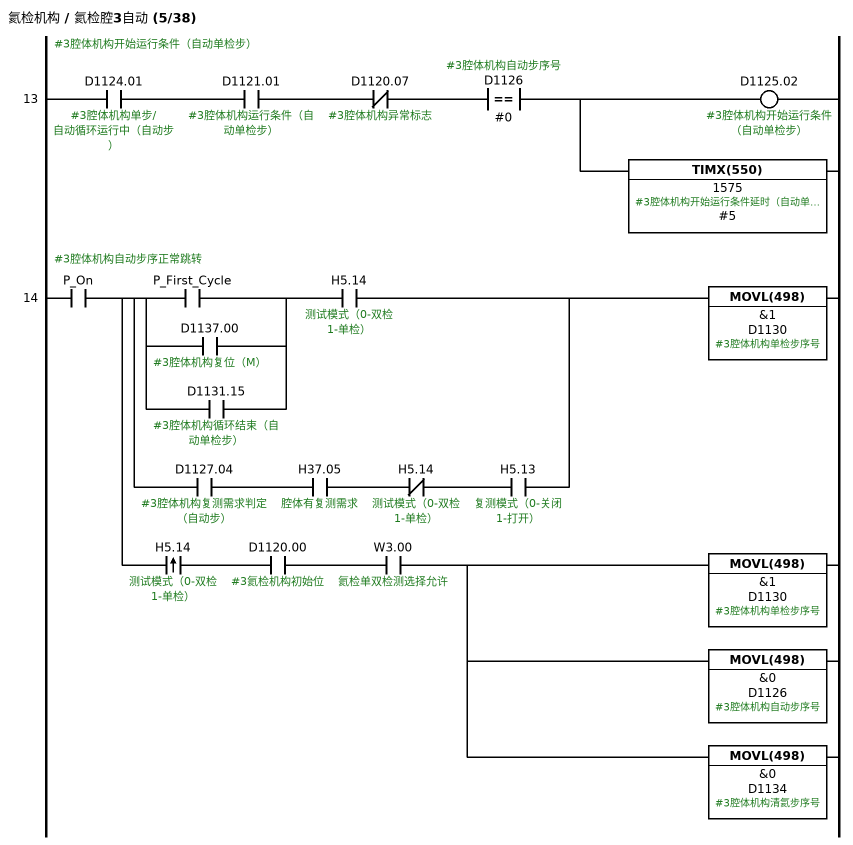
; [picture p288: 氦检机构 / 氦检腔3自动, rungs 13-14]
; rung 13: #3腔体机构开始运行条件（自动单检步）
LD D1124.01  ; #3腔体机构单步/自动循环运行中（自动步）
AND D1121.01  ; #3腔体机构运行条件（自动单检步）
ANDNOT D1120.07  ; #3腔体机构异常标志
AND=L(301) D1126 #0  ; #3腔体机构自动步序号
OUT D1125.02  ; #3腔体机构开始运行条件（自动单检步）
TIMX(550) 1575 #5  ; #3腔体机构开始运行条件延时（自动单检步）
; rung 14: #3腔体机构自动步序正常跳转
LD P_On
OUT TR0
LD P_First_Cycle
OR D1137.00  ; #3腔体机构复位（M）
OR D1131.15  ; #3腔体机构循环结束（自动单检步）
AND H5.14  ; 测试模式（0-双检 1-单检）
LD D1127.04  ; #3腔体机构复测需求判定（自动步）
AND H37.05  ; 腔体有复测需求
ANDNOT H5.14  ; 测试模式（0-双检 1-单检）
AND H5.13  ; 复测模式（0-关闭 1-打开）
ORLD
ANDLD
MOVL(498) &1 D1130  ; #3腔体机构单检步序号
LD TR0
@AND H5.14  ; 测试模式（0-双检 1-单检）
AND D1120.00  ; #3氦检机构初始位
AND W3.00  ; 氦检单双检测选择允许
MOVL(498) &1 D1130  ; #3腔体机构单检步序号
MOVL(498) &0 D1126  ; #3腔体机构自动步序号
MOVL(498) &0 D1134  ; #3腔体机构清氦步序号

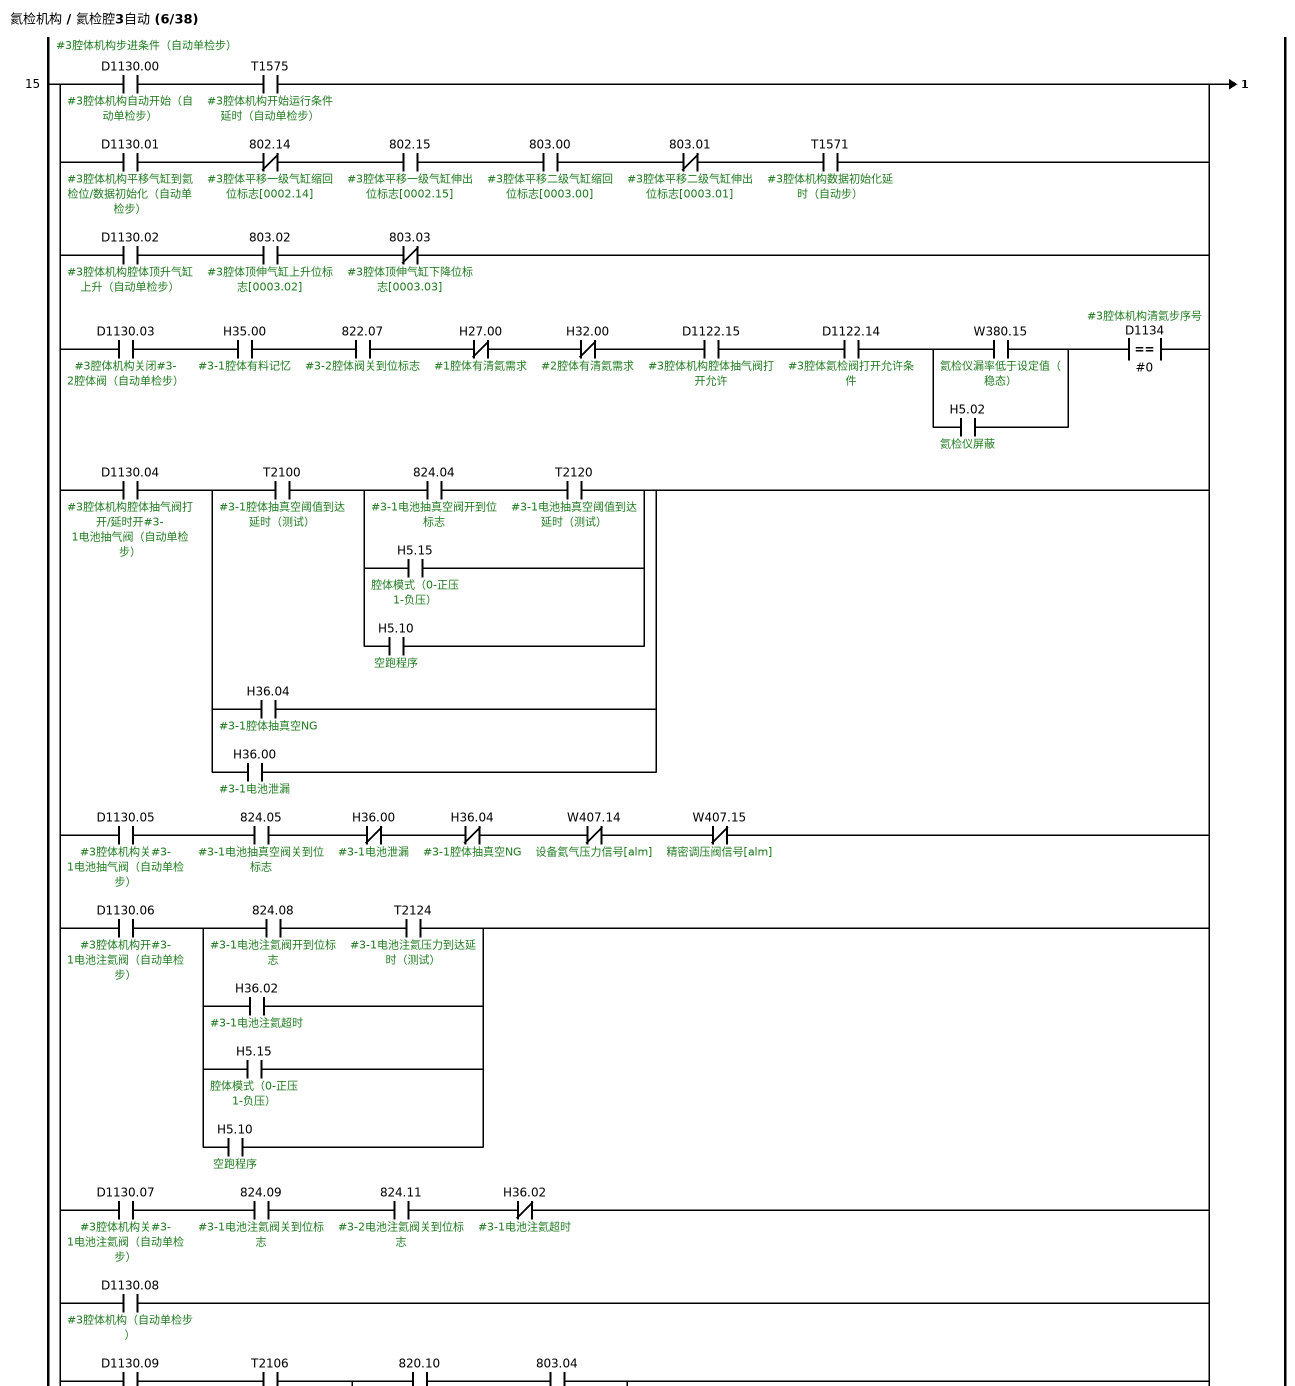

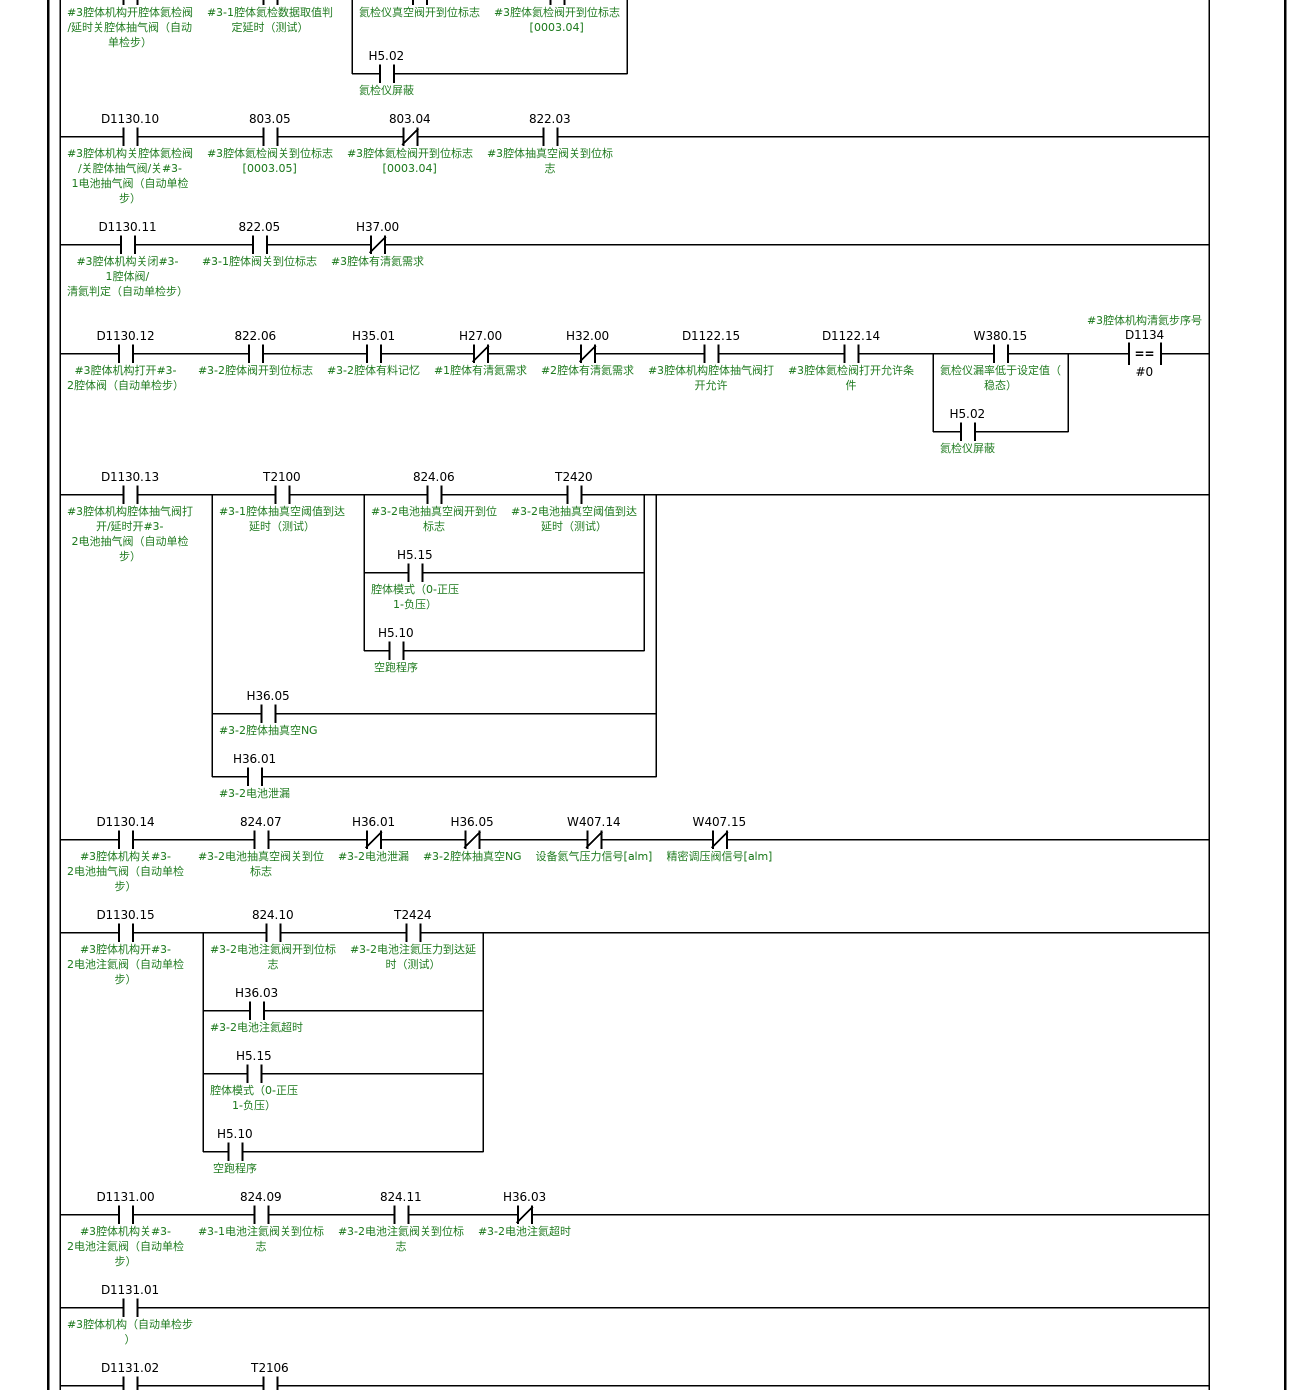

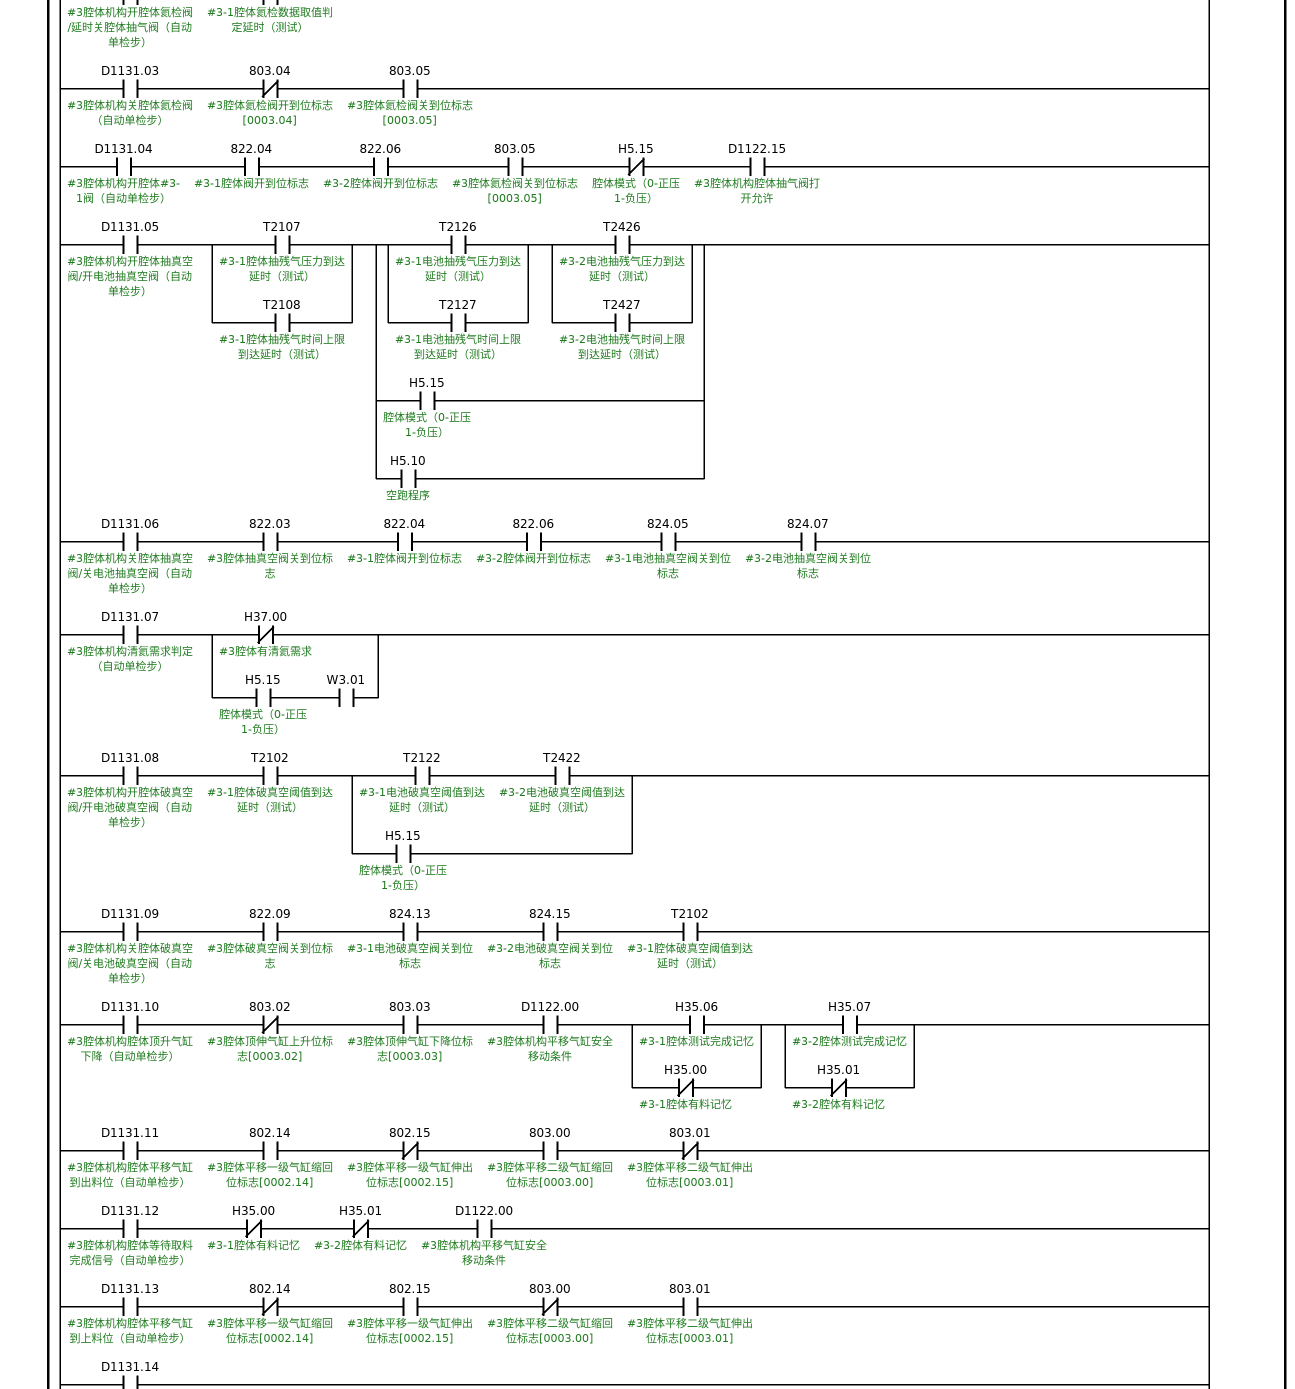

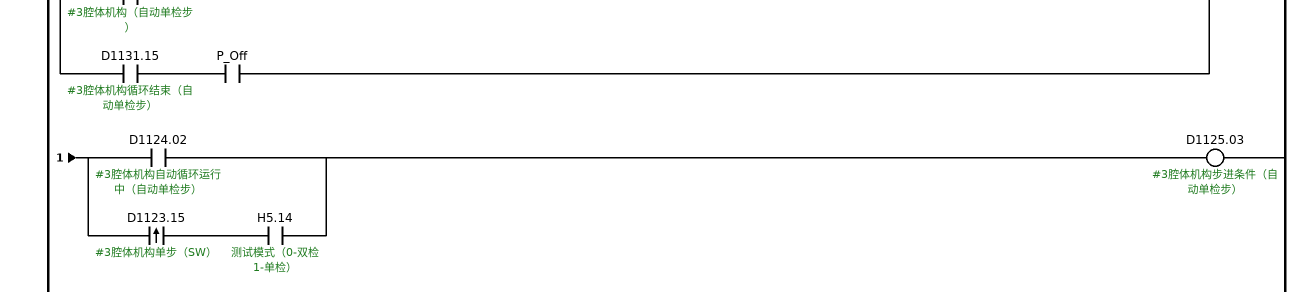
; rung 15: #3腔体机构步进条件（自动单检步）
LD D1130.00  ; #3腔体机构自动开始（自动单检步）
AND T1575  ; #3腔体机构开始运行条件延时（自动单检步）
LD D1130.01  ; #3腔体机构平移气缸到氦检位/数据初始化（自动单检步）
ANDNOT 802.14  ; #3腔体平移一级气缸缩回位标志[0002.14]
AND 802.15  ; #3腔体平移一级气缸伸出位标志[0002.15]
AND 803.00  ; #3腔体平移二级气缸缩回位标志[0003.00]
ANDNOT 803.01  ; #3腔体平移二级气缸伸出位标志[0003.01]
AND T1571  ; #3腔体机构数据初始化延时（自动步）
ORLD
LD D1130.02  ; #3腔体机构腔体顶升气缸上升（自动单检步）
AND 803.02  ; #3腔体顶伸气缸上升位标志[0003.02]
ANDNOT 803.03  ; #3腔体顶伸气缸下降位标志[0003.03]
ORLD
LD D1130.03  ; #3腔体机构关闭#3-2腔体阀（自动单检步）
AND H35.00  ; #3-1腔体有料记忆
AND 822.07  ; #3-2腔体阀关到位标志
ANDNOT H27.00  ; #1腔体有清氦需求
ANDNOT H32.00  ; #2腔体有清氦需求
AND D1122.15  ; #3腔体机构腔体抽气阀打开允许
AND D1122.14  ; #3腔体氦检阀打开允许条件
LD W380.15  ; 氦检仪漏率低于设定值（稳态）
OR H5.02  ; 氦检仪屏蔽
ANDLD
AND=L(301) D1134 #0  ; #3腔体机构清氦步序号
ORLD
LD D1130.04  ; #3腔体机构腔体抽气阀打开/延时开#3-1电池抽气阀（自动单检步）
LD T2100  ; #3-1腔体抽真空阈值到达延时（测试）
LD 824.04  ; #3-1电池抽真空阀开到位标志
AND T2120  ; #3-1电池抽真空阈值到达延时（测试）
OR H5.15  ; 腔体模式（0-正压 1-负压）
OR H5.10  ; 空跑程序
ANDLD
OR H36.04  ; #3-1腔体抽真空NG
OR H36.00  ; #3-1电池泄漏
ANDLD
ORLD
LD D1130.05  ; #3腔体机构关#3-1电池抽气阀（自动单检步）
AND 824.05  ; #3-1电池抽真空阀关到位标志
ANDNOT H36.00  ; #3-1电池泄漏
ANDNOT H36.04  ; #3-1腔体抽真空NG
ANDNOT W407.14  ; 设备氦气压力信号[alm]
ANDNOT W407.15  ; 精密调压阀信号[alm]
ORLD
LD D1130.06  ; #3腔体机构开#3-1电池注氦阀（自动单检步）
LD 824.08  ; #3-1电池注氦阀开到位标志
AND T2124  ; #3-1电池注氦压力到达延时（测试）
OR H36.02  ; #3-1电池注氦超时
OR H5.15  ; 腔体模式（0-正压 1-负压）
OR H5.10  ; 空跑程序
ANDLD
ORLD
LD D1130.07  ; #3腔体机构关#3-1电池注氦阀（自动单检步）
AND 824.09  ; #3-1电池注氦阀关到位标志
AND 824.11  ; #3-2电池注氦阀关到位标志
ANDNOT H36.02  ; #3-1电池注氦超时
ORLD
OR D1130.08  ; #3腔体机构（自动单检步）
LD D1130.09  ; #3腔体机构开腔体氦检阀/延时关腔体抽气阀（自动单检步）
AND T2106  ; #3-1腔体氦检数据取值判定延时（测试）
LD 820.10  ; 氦检仪真空阀开到位标志
AND 803.04  ; #3腔体氦检阀开到位标志[0003.04]
OR H5.02  ; 氦检仪屏蔽
ANDLD
ORLD
LD D1130.10  ; #3腔体机构关腔体氦检阀/关腔体抽气阀/关#3-1电池抽气阀（自动单检步）
AND 803.05  ; #3腔体氦检阀关到位标志[0003.05]
ANDNOT 803.04  ; #3腔体氦检阀开到位标志[0003.04]
AND 822.03  ; #3腔体抽真空阀关到位标志
ORLD
LD D1130.11  ; #3腔体机构关闭#3-1腔体阀/清氦判定（自动单检步）
AND 822.05  ; #3-1腔体阀关到位标志
ANDNOT H37.00  ; #3腔体有清氦需求
ORLD
LD D1130.12  ; #3腔体机构打开#3-2腔体阀（自动单检步）
AND 822.06  ; #3-2腔体阀开到位标志
AND H35.01  ; #3-2腔体有料记忆
ANDNOT H27.00  ; #1腔体有清氦需求
ANDNOT H32.00  ; #2腔体有清氦需求
AND D1122.15  ; #3腔体机构腔体抽气阀打开允许
AND D1122.14  ; #3腔体氦检阀打开允许条件
LD W380.15  ; 氦检仪漏率低于设定值（稳态）
OR H5.02  ; 氦检仪屏蔽
ANDLD
AND=L(301) D1134 #0  ; #3腔体机构清氦步序号
ORLD
LD D1130.13  ; #3腔体机构腔体抽气阀打开/延时开#3-2电池抽气阀（自动单检步）
LD T2100  ; #3-1腔体抽真空阈值到达延时（测试）
LD 824.06  ; #3-2电池抽真空阀开到位标志
AND T2420  ; #3-2电池抽真空阈值到达延时（测试）
OR H5.15  ; 腔体模式（0-正压 1-负压）
OR H5.10  ; 空跑程序
ANDLD
OR H36.05  ; #3-2腔体抽真空NG
OR H36.01  ; #3-2电池泄漏
ANDLD
ORLD
LD D1130.14  ; #3腔体机构关#3-2电池抽气阀（自动单检步）
AND 824.07  ; #3-2电池抽真空阀关到位标志
ANDNOT H36.01  ; #3-2电池泄漏
ANDNOT H36.05  ; #3-2腔体抽真空NG
ANDNOT W407.14  ; 设备氦气压力信号[alm]
ANDNOT W407.15  ; 精密调压阀信号[alm]
ORLD
LD D1130.15  ; #3腔体机构开#3-2电池注氦阀（自动单检步）
LD 824.10  ; #3-2电池注氦阀开到位标志
AND T2424  ; #3-2电池注氦压力到达延时（测试）
OR H36.03  ; #3-2电池注氦超时
OR H5.15  ; 腔体模式（0-正压 1-负压）
OR H5.10  ; 空跑程序
ANDLD
ORLD
LD D1131.00  ; #3腔体机构关#3-2电池注氦阀（自动单检步）
AND 824.09  ; #3-1电池注氦阀关到位标志
AND 824.11  ; #3-2电池注氦阀关到位标志
ANDNOT H36.03  ; #3-2电池注氦超时
ORLD
OR D1131.01  ; #3腔体机构（自动单检步）
LD D1131.02  ; #3腔体机构开腔体氦检阀/延时关腔体抽气阀（自动单检步）
AND T2106  ; #3-1腔体氦检数据取值判定延时（测试）
ORLD
LD D1131.03  ; #3腔体机构关腔体氦检阀（自动单检步）
ANDNOT 803.04  ; #3腔体氦检阀开到位标志[0003.04]
AND 803.05  ; #3腔体氦检阀关到位标志[0003.05]
ORLD
LD D1131.04  ; #3腔体机构开腔体#3-1阀（自动单检步）
AND 822.04  ; #3-1腔体阀开到位标志
AND 822.06  ; #3-2腔体阀开到位标志
AND 803.05  ; #3腔体氦检阀关到位标志[0003.05]
ANDNOT H5.15  ; 腔体模式（0-正压 1-负压）
AND D1122.15  ; #3腔体机构腔体抽气阀打开允许
ORLD
LD D1131.05  ; #3腔体机构开腔体抽真空阀/开电池抽真空阀（自动单检步）
LD T2107  ; #3-1腔体抽残气压力到达延时（测试）
OR T2108  ; #3-1腔体抽残气时间上限到达延时（测试）
ANDLD
LD T2126  ; #3-1电池抽残气压力到达延时（测试）
OR T2127  ; #3-1电池抽残气时间上限到达延时（测试）
LD T2426  ; #3-2电池抽残气压力到达延时（测试）
OR T2427  ; #3-2电池抽残气时间上限到达延时（测试）
ANDLD
OR H5.15  ; 腔体模式（0-正压 1-负压）
OR H5.10  ; 空跑程序
ANDLD
ORLD
LD D1131.06  ; #3腔体机构关腔体抽真空阀/关电池抽真空阀（自动单检步）
AND 822.03  ; #3腔体抽真空阀关到位标志
AND 822.04  ; #3-1腔体阀开到位标志
AND 822.06  ; #3-2腔体阀开到位标志
AND 824.05  ; #3-1电池抽真空阀关到位标志
AND 824.07  ; #3-2电池抽真空阀关到位标志
ORLD
LD D1131.07  ; #3腔体机构清氦需求判定（自动单检步）
LDNOT H37.00  ; #3腔体有清氦需求
LD H5.15  ; 腔体模式（0-正压 1-负压）
AND W3.01
ORLD
ANDLD
ORLD
LD D1131.08  ; #3腔体机构开腔体破真空阀/开电池破真空阀（自动单检步）
AND T2102  ; #3-1腔体破真空阈值到达延时（测试）
LD T2122  ; #3-1电池破真空阈值到达延时（测试）
AND T2422  ; #3-2电池破真空阈值到达延时（测试）
OR H5.15  ; 腔体模式（0-正压 1-负压）
ANDLD
ORLD
LD D1131.09  ; #3腔体机构关腔体破真空阀/关电池破真空阀（自动单检步）
AND 822.09  ; #3腔体破真空阀关到位标志
AND 824.13  ; #3-1电池破真空阀关到位标志
AND 824.15  ; #3-2电池破真空阀关到位标志
AND T2102  ; #3-1腔体破真空阈值到达延时（测试）
ORLD
LD D1131.10  ; #3腔体机构腔体顶升气缸下降（自动单检步）
ANDNOT 803.02  ; #3腔体顶伸气缸上升位标志[0003.02]
AND 803.03  ; #3腔体顶伸气缸下降位标志[0003.03]
AND D1122.00  ; #3腔体机构平移气缸安全移动条件
LD H35.06  ; #3-1腔体测试完成记忆
ORNOT H35.00  ; #3-1腔体有料记忆
ANDLD
LD H35.07  ; #3-2腔体测试完成记忆
ORNOT H35.01  ; #3-2腔体有料记忆
ANDLD
ORLD
LD D1131.11  ; #3腔体机构腔体平移气缸到出料位（自动单检步）
AND 802.14  ; #3腔体平移一级气缸缩回位标志[0002.14]
ANDNOT 802.15  ; #3腔体平移一级气缸伸出位标志[0002.15]
AND 803.00  ; #3腔体平移二级气缸缩回位标志[0003.00]
ANDNOT 803.01  ; #3腔体平移二级气缸伸出位标志[0003.01]
ORLD
LD D1131.12  ; #3腔体机构腔体等待取料完成信号（自动单检步）
ANDNOT H35.00  ; #3-1腔体有料记忆
ANDNOT H35.01  ; #3-2腔体有料记忆
AND D1122.00  ; #3腔体机构平移气缸安全移动条件
ORLD
LD D1131.13  ; #3腔体机构腔体平移气缸到上料位（自动单检步）
ANDNOT 802.14  ; #3腔体平移一级气缸缩回位标志[0002.14]
AND 802.15  ; #3腔体平移一级气缸伸出位标志[0002.15]
ANDNOT 803.00  ; #3腔体平移二级气缸缩回位标志[0003.00]
AND 803.01  ; #3腔体平移二级气缸伸出位标志[0003.01]
ORLD
OR D1131.14  ; #3腔体机构（自动单检步）
LD D1131.15  ; #3腔体机构循环结束（自动单检步）
AND P_Off
ORLD
LD D1124.02  ; #3腔体机构自动循环运行中（自动单检步）
@LD D1123.15  ; #3腔体机构单步（SW）
AND H5.14  ; 测试模式（0-双检 1-单检）
ORLD
ANDLD
OUT D1125.03  ; #3腔体机构步进条件（自动单检步）

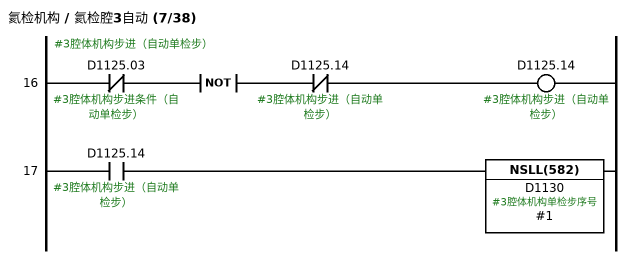
; rung 16: #3腔体机构步进（自动单检步）
LDNOT D1125.03  ; #3腔体机构步进条件（自动单检步）
NOT(520)
ANDNOT D1125.14  ; #3腔体机构步进（自动单检步）
OUT D1125.14  ; #3腔体机构步进（自动单检步）
; rung 17
LD D1125.14  ; #3腔体机构步进（自动单检步）
NSLL(582) D1130 #1  ; #3腔体机构单检步序号

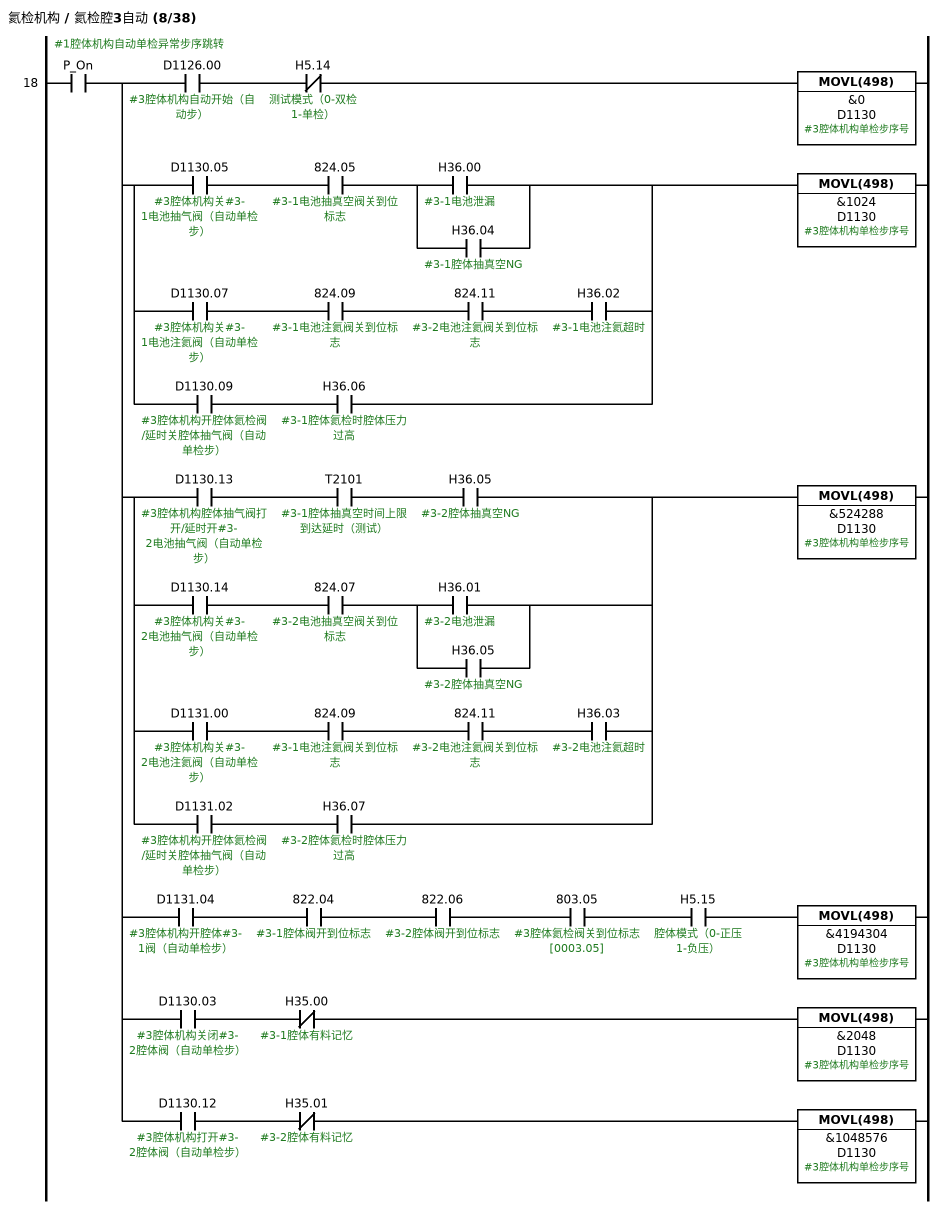
; rung 18: #1腔体机构自动单检异常步序跳转
LD P_On
OUT TR0
AND D1126.00  ; #3腔体机构自动开始（自动步）
ANDNOT H5.14  ; 测试模式（0-双检 1-单检）
MOVL(498) &0 D1130  ; #3腔体机构单检步序号
LD TR0
LD D1130.05  ; #3腔体机构关#3-1电池抽气阀（自动单检步）
AND 824.05  ; #3-1电池抽真空阀关到位标志
LD H36.00  ; #3-1电池泄漏
OR H36.04  ; #3-1腔体抽真空NG
ANDLD
LD D1130.07  ; #3腔体机构关#3-1电池注氦阀（自动单检步）
AND 824.09  ; #3-1电池注氦阀关到位标志
AND 824.11  ; #3-2电池注氦阀关到位标志
AND H36.02  ; #3-1电池注氦超时
ORLD
LD D1130.09  ; #3腔体机构开腔体氦检阀/延时关腔体抽气阀（自动单检步）  // 氦检阀开启后腔体压力超过安全阀值，测试判定为NG（氦检异常）
AND H36.06  ; #3-1腔体氦检时腔体压力过高
ORLD
ANDLD
MOVL(498) &1024 D1130  ; #3腔体机构单检步序号  // #1-1腔体出现腔体泄漏，电池泄漏，注氦超时的情况，均跳转至单检步序D1070.10
LD TR0
LD D1130.13  ; #3腔体机构腔体抽气阀打开/延时开#3-2电池抽气阀（自动单检步）
AND T2101  ; #3-1腔体抽真空时间上限到达延时（测试）
AND H36.05  ; #3-2腔体抽真空NG
LD D1130.14  ; #3腔体机构关#3-2电池抽气阀（自动单检步）
AND 824.07  ; #3-2电池抽真空阀关到位标志
LD H36.01  ; #3-2电池泄漏
OR H36.05  ; #3-2腔体抽真空NG
ANDLD
ORLD
LD D1131.00  ; #3腔体机构关#3-2电池注氦阀（自动单检步）
AND 824.09  ; #3-1电池注氦阀关到位标志
AND 824.11  ; #3-2电池注氦阀关到位标志
AND H36.03  ; #3-2电池注氦超时
ORLD
LD D1131.02  ; #3腔体机构开腔体氦检阀/延时关腔体抽气阀（自动单检步）  // 氦检阀开启后腔体压力超过安全阀值，测试判定为NG（氦检异常）
AND H36.07  ; #3-2腔体氦检时腔体压力过高
ORLD
ANDLD
MOVL(498) &524288 D1130  ; #3腔体机构单检步序号  // #1-2腔体出现腔体泄漏，电池泄漏，注氦超时的情况，均跳转至单检步序D1071.03
LD TR0
AND D1131.04  ; #3腔体机构开腔体#3-1阀（自动单检步）
AND 822.04  ; #3-1腔体阀开到位标志
AND 822.06  ; #3-2腔体阀开到位标志
AND 803.05  ; #3腔体氦检阀关到位标志[0003.05]
AND H5.15  ; 腔体模式（0-正压 1-负压）
MOVL(498) &4194304 D1130  ; #3腔体机构单检步序号  // 负压模式下步序正常流程步序不需要抽残气，直接跳转至D1071.06
LD TR0
AND D1130.03  ; #3腔体机构关闭#3-2腔体阀（自动单检步）
ANDNOT H35.00  ; #3-1腔体有料记忆
MOVL(498) &2048 D1130  ; #3腔体机构单检步序号  // 清尾料是#1-1无料，跳转至D1070.11
LD TR0
AND D1130.12  ; #3腔体机构打开#3-2腔体阀（自动单检步）
ANDNOT H35.01  ; #3-2腔体有料记忆
MOVL(498) &1048576 D1130  ; #3腔体机构单检步序号  // 清尾料时#1-2无料，跳转至D1071.04
; rung 19: ******************************* / 清氦步序 / *******************************

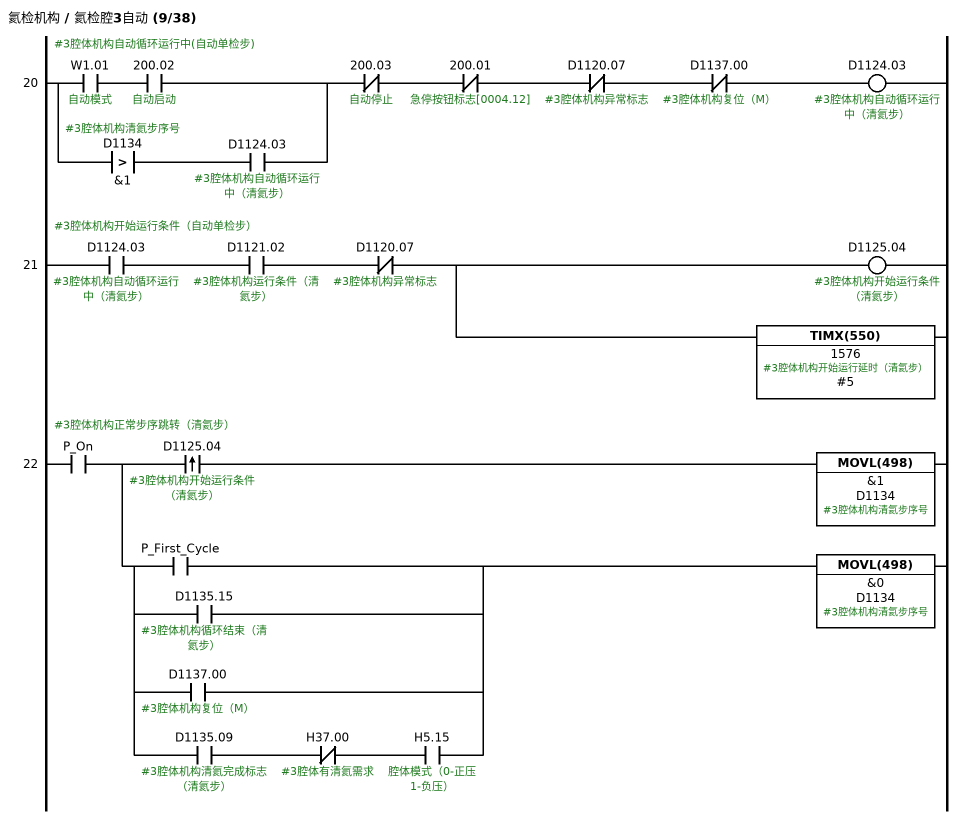
; rung 20: #3腔体机构自动循环运行中(自动单检步)
LD W1.01  ; 自动模式
AND 200.02  ; 自动启动
LD>L(321) D1134 &1  ; #3腔体机构清氦步序号
AND D1124.03  ; #3腔体机构自动循环运行中（清氦步）
ORLD
ANDNOT 200.03  ; 自动停止
ANDNOT 200.01  ; 急停按钮标志[0004.12]
ANDNOT D1120.07  ; #3腔体机构异常标志
ANDNOT D1137.00  ; #3腔体机构复位（M）
OUT D1124.03  ; #3腔体机构自动循环运行中（清氦步）
; rung 21: #3腔体机构开始运行条件（自动单检步）
LD D1124.03  ; #3腔体机构自动循环运行中（清氦步）
AND D1121.02  ; #3腔体机构运行条件（清氦步）
ANDNOT D1120.07  ; #3腔体机构异常标志
OUT D1125.04  ; #3腔体机构开始运行条件（清氦步）
TIMX(550) 1576 #5  ; #3腔体机构开始运行延时（清氦步）
; rung 22: #3腔体机构正常步序跳转（清氦步）
LD P_On
OUT TR0
@AND D1125.04  ; #3腔体机构开始运行条件（清氦步）
MOVL(498) &1 D1134  ; #3腔体机构清氦步序号
LD TR0
LD P_First_Cycle
OR D1135.15  ; #3腔体机构循环结束（清氦步）
OR D1137.00  ; #3腔体机构复位（M）
LD D1135.09  ; #3腔体机构清氦完成标志（清氦步）  // 正压腔体是待料清氦，需跳转回测试步序
ANDNOT H37.00  ; #3腔体有清氦需求
AND H5.15  ; 腔体模式（0-正压 1-负压）
ORLD
ANDLD
MOVL(498) &0 D1134  ; #3腔体机构清氦步序号

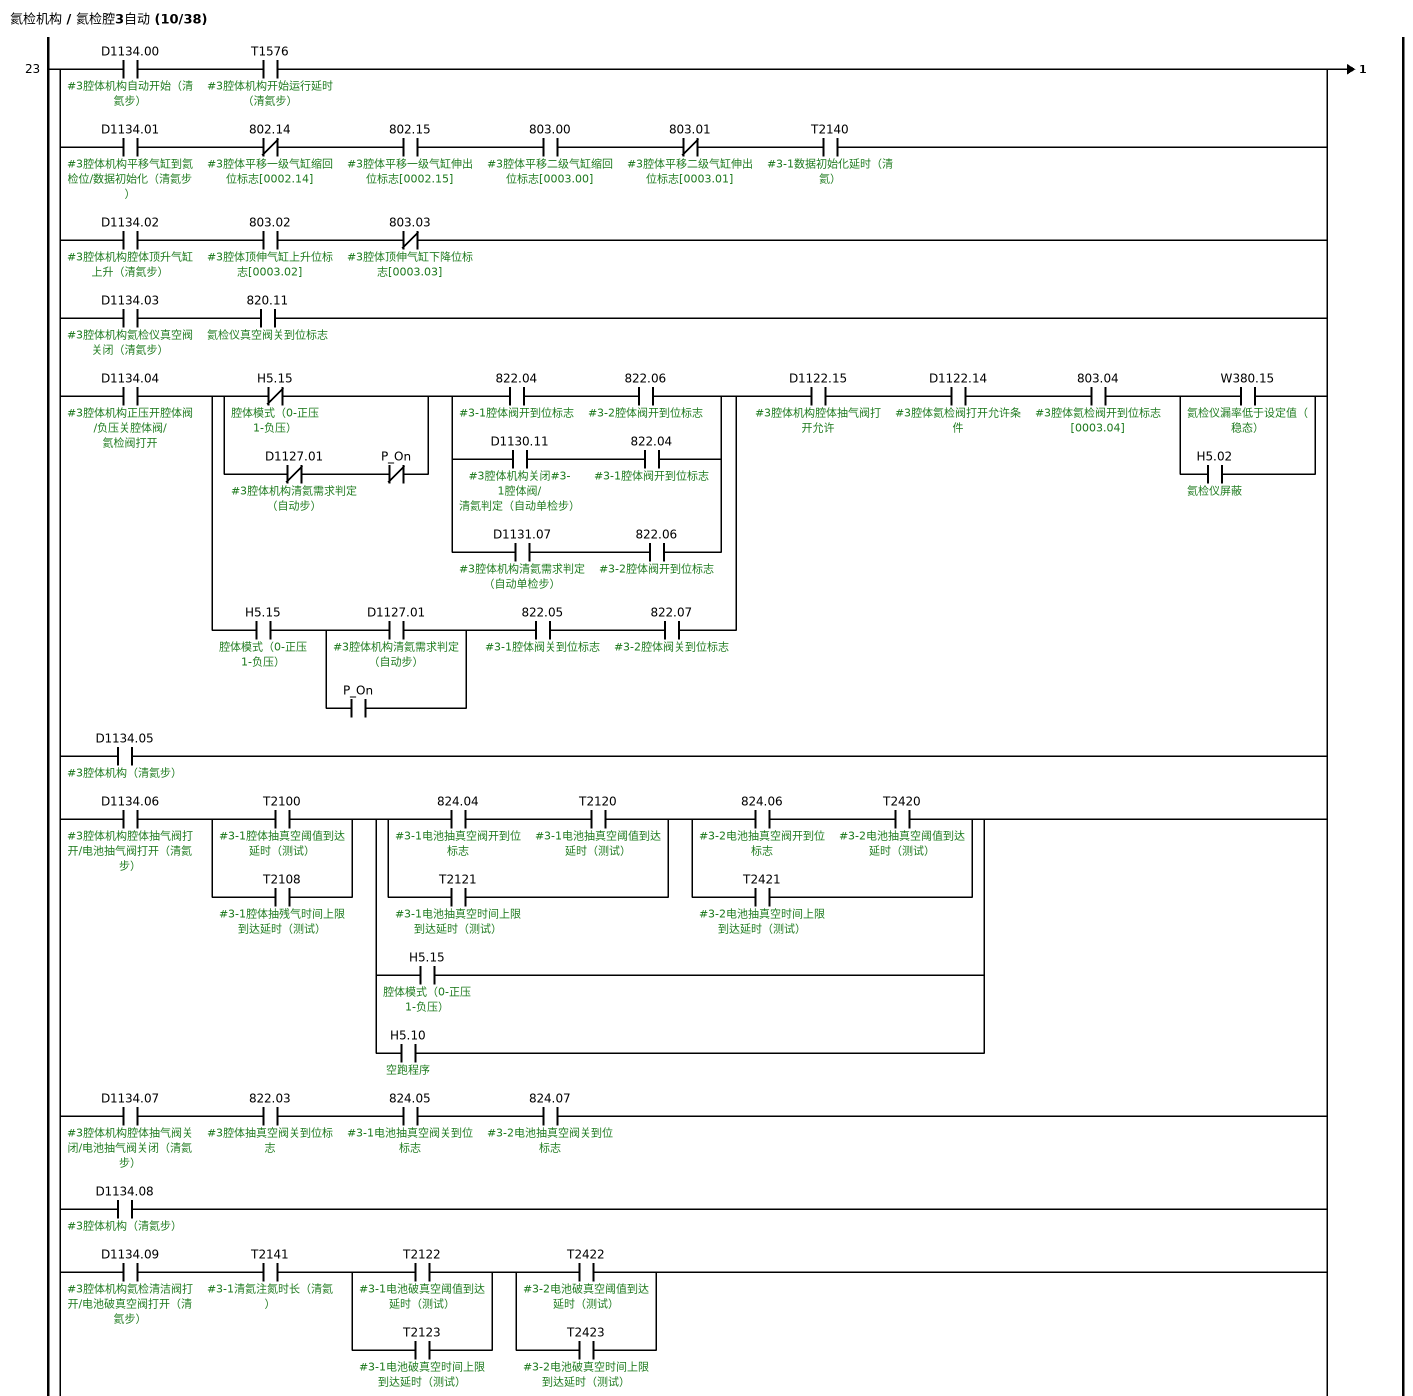

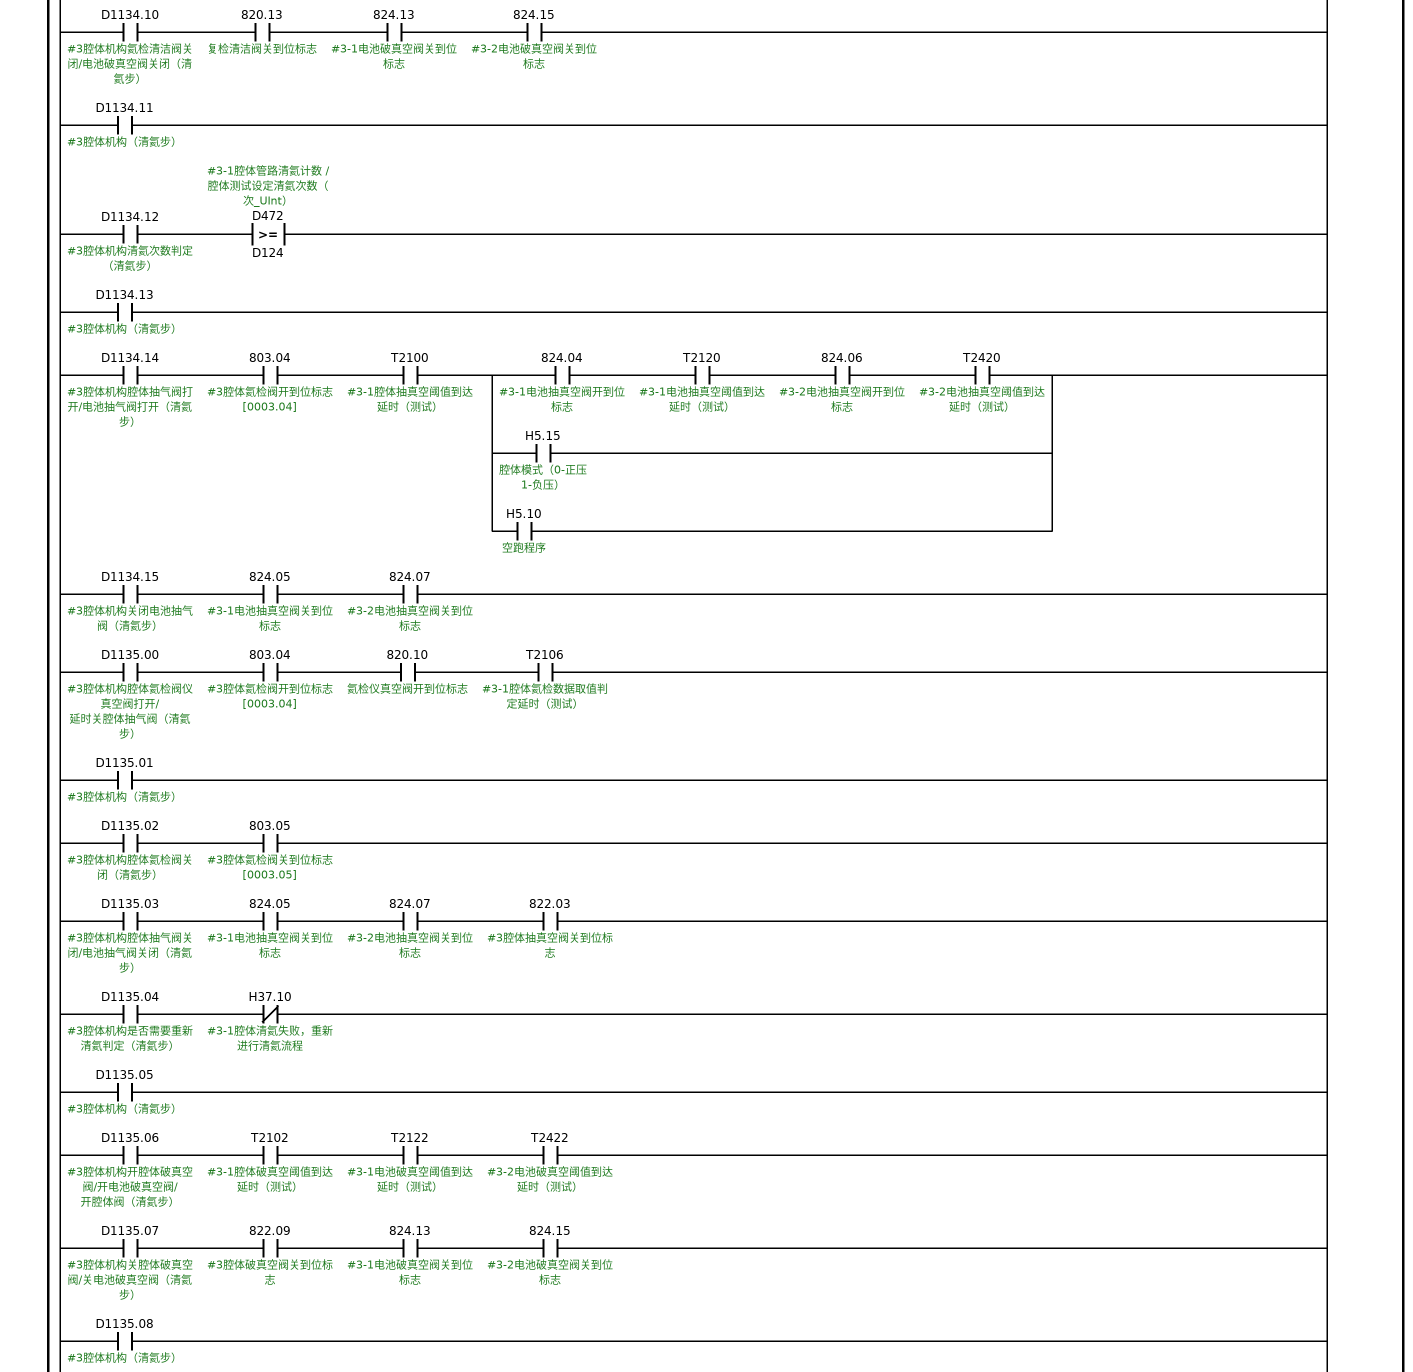

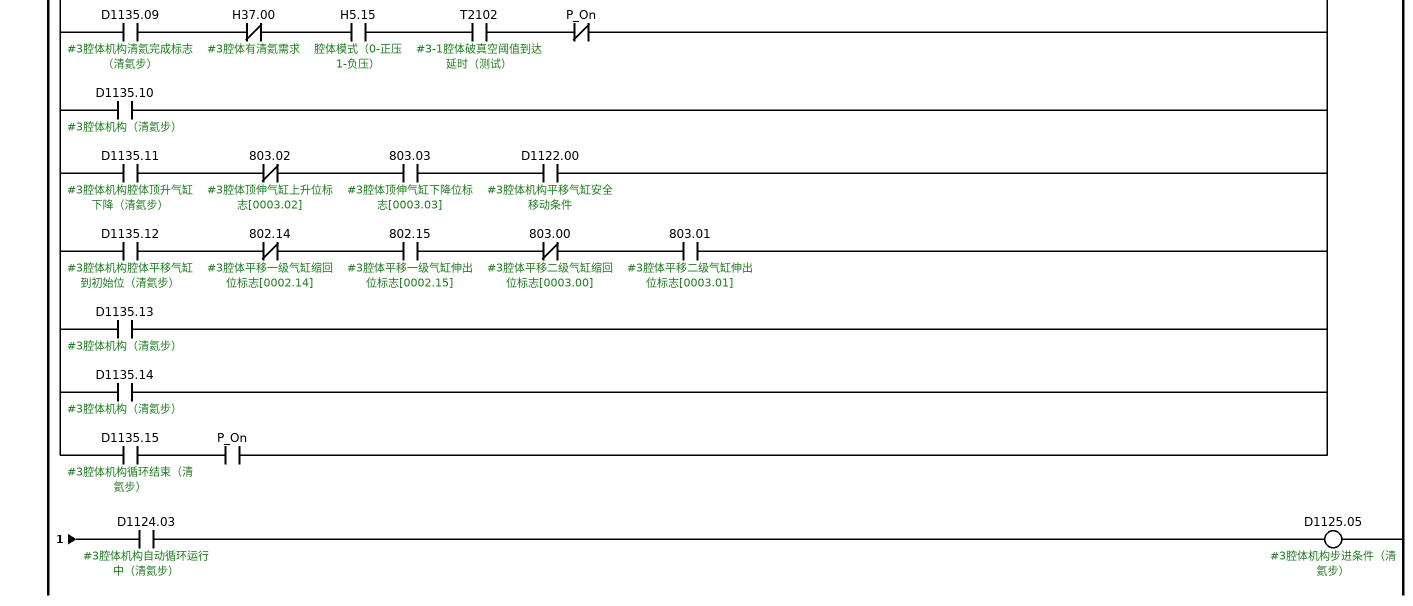
; rung 23
LD D1134.00  ; #3腔体机构自动开始（清氦步）
AND T1576  ; #3腔体机构开始运行延时（清氦步）
LD D1134.01  ; #3腔体机构平移气缸到氦检位/数据初始化（清氦步）
ANDNOT 802.14  ; #3腔体平移一级气缸缩回位标志[0002.14]
AND 802.15  ; #3腔体平移一级气缸伸出位标志[0002.15]
AND 803.00  ; #3腔体平移二级气缸缩回位标志[0003.00]
ANDNOT 803.01  ; #3腔体平移二级气缸伸出位标志[0003.01]
AND T2140  ; #3-1数据初始化延时（清氦）
ORLD
LD D1134.02  ; #3腔体机构腔体顶升气缸上升（清氦步）
AND 803.02  ; #3腔体顶伸气缸上升位标志[0003.02]
ANDNOT 803.03  ; #3腔体顶伸气缸下降位标志[0003.03]
ORLD
LD D1134.03  ; #3腔体机构氦检仪真空阀关闭（清氦步）
AND 820.11  ; 氦检仪真空阀关到位标志
ORLD
LD D1134.04  ; #3腔体机构正压开腔体阀/负压关腔体阀/氦检阀打开  // 负压模式下，复测前的清氦不允许抽电池
LDNOT H5.15  ; 腔体模式（0-正压 1-负压）
LDNOT D1127.01  ; #3腔体机构清氦需求判定（自动步）
ANDNOT P_On
ORLD
LD 822.04  ; #3-1腔体阀开到位标志
AND 822.06  ; #3-2腔体阀开到位标志
LD D1130.11  ; #3腔体机构关闭#3-1腔体阀/清氦判定（自动单检步）
AND 822.04  ; #3-1腔体阀开到位标志
ORLD
LD D1131.07  ; #3腔体机构清氦需求判定（自动单检步）
AND 822.06  ; #3-2腔体阀开到位标志
ORLD
ANDLD
LD H5.15  ; 腔体模式（0-正压 1-负压）
LD D1127.01  ; #3腔体机构清氦需求判定（自动步）
OR P_On
ANDLD
AND 822.05  ; #3-1腔体阀关到位标志
AND 822.07  ; #3-2腔体阀关到位标志
ORLD
ANDLD
AND D1122.15  ; #3腔体机构腔体抽气阀打开允许
AND D1122.14  ; #3腔体氦检阀打开允许条件
AND 803.04  ; #3腔体氦检阀开到位标志[0003.04]
LD W380.15  ; 氦检仪漏率低于设定值（稳态）
OR H5.02  ; 氦检仪屏蔽
ANDLD
ORLD
OR D1134.05  ; #3腔体机构（清氦步）
LD D1134.06  ; #3腔体机构腔体抽气阀打开/电池抽气阀打开（清氦步）
LD T2100  ; #3-1腔体抽真空阈值到达延时（测试）
OR T2108  ; #3-1腔体抽残气时间上限到达延时（测试）
ANDLD
LD 824.04  ; #3-1电池抽真空阀开到位标志
AND T2120  ; #3-1电池抽真空阈值到达延时（测试）
OR T2121  ; #3-1电池抽真空时间上限到达延时（测试）
LD 824.06  ; #3-2电池抽真空阀开到位标志
AND T2420  ; #3-2电池抽真空阈值到达延时（测试）
OR T2421  ; #3-2电池抽真空时间上限到达延时（测试）
ANDLD
OR H5.15  ; 腔体模式（0-正压 1-负压）
OR H5.10  ; 空跑程序
ANDLD
ORLD
LD D1134.07  ; #3腔体机构腔体抽气阀关闭/电池抽气阀关闭（清氦步）
AND 822.03  ; #3腔体抽真空阀关到位标志
AND 824.05  ; #3-1电池抽真空阀关到位标志
AND 824.07  ; #3-2电池抽真空阀关到位标志
ORLD
OR D1134.08  ; #3腔体机构（清氦步）
LD D1134.09  ; #3腔体机构氦检清洁阀打开/电池破真空阀打开（清氦步）
AND T2141  ; #3-1清氦注氮时长（清氦）
LD T2122  ; #3-1电池破真空阈值到达延时（测试）
OR T2123  ; #3-1电池破真空时间上限到达延时（测试）
ANDLD
LD T2422  ; #3-2电池破真空阈值到达延时（测试）
OR T2423  ; #3-2电池破真空时间上限到达延时（测试）
ANDLD
ORLD
LD D1134.10  ; #3腔体机构氦检清洁阀关闭/电池破真空阀关闭（清氦步）
AND 820.13  ; 复检清洁阀关到位标志
AND 824.13  ; #3-1电池破真空阀关到位标志
AND 824.15  ; #3-2电池破真空阀关到位标志
ORLD
OR D1134.11  ; #3腔体机构（清氦步）
LD D1134.12  ; #3腔体机构清氦次数判定（清氦步）
AND>=(325) D472 D124  ; #3-1腔体管路清氦计数, 腔体测试设定清氦次数（次_UInt）
ORLD
OR D1134.13  ; #3腔体机构（清氦步）
LD D1134.14  ; #3腔体机构腔体抽气阀打开/电池抽气阀打开（清氦步）
AND 803.04  ; #3腔体氦检阀开到位标志[0003.04]
AND T2100  ; #3-1腔体抽真空阈值到达延时（测试）
LD 824.04  ; #3-1电池抽真空阀开到位标志
AND T2120  ; #3-1电池抽真空阈值到达延时（测试）
AND 824.06  ; #3-2电池抽真空阀开到位标志
AND T2420  ; #3-2电池抽真空阈值到达延时（测试）
OR H5.15  ; 腔体模式（0-正压 1-负压）
OR H5.10  ; 空跑程序
ANDLD
ORLD
LD D1134.15  ; #3腔体机构关闭电池抽气阀（清氦步）
AND 824.05  ; #3-1电池抽真空阀关到位标志
AND 824.07  ; #3-2电池抽真空阀关到位标志
ORLD
LD D1135.00  ; #3腔体机构腔体氦检阀仪真空阀打开/延时关腔体抽气阀（清氦步）
AND 803.04  ; #3腔体氦检阀开到位标志[0003.04]
AND 820.10  ; 氦检仪真空阀开到位标志
AND T2106  ; #3-1腔体氦检数据取值判定延时（测试）
ORLD
OR D1135.01  ; #3腔体机构（清氦步）
LD D1135.02  ; #3腔体机构腔体氦检阀关闭（清氦步）
AND 803.05  ; #3腔体氦检阀关到位标志[0003.05]
ORLD
LD D1135.03  ; #3腔体机构腔体抽气阀关闭/电池抽气阀关闭（清氦步）
AND 824.05  ; #3-1电池抽真空阀关到位标志
AND 824.07  ; #3-2电池抽真空阀关到位标志
AND 822.03  ; #3腔体抽真空阀关到位标志
ORLD
LD D1135.04  ; #3腔体机构是否需要重新清氦判定（清氦步）
ANDNOT H37.10  ; #3-1腔体清氦失败，重新进行清氦流程  // 清氦失败，重新进行清氦
ORLD
OR D1135.05  ; #3腔体机构（清氦步）
LD D1135.06  ; #3腔体机构开腔体破真空阀/开电池破真空阀/开腔体阀（清氦步）
AND T2102  ; #3-1腔体破真空阈值到达延时（测试）
AND T2122  ; #3-1电池破真空阈值到达延时（测试）
AND T2422  ; #3-2电池破真空阈值到达延时（测试）
ORLD
LD D1135.07  ; #3腔体机构关腔体破真空阀/关电池破真空阀（清氦步）
AND 822.09  ; #3腔体破真空阀关到位标志
AND 824.13  ; #3-1电池破真空阀关到位标志
AND 824.15  ; #3-2电池破真空阀关到位标志
ORLD
OR D1135.08  ; #3腔体机构（清氦步）
LD D1135.09  ; #3腔体机构清氦完成标志（清氦步）  // 正压腔体是待料清氦，需跳转回测试步序
ANDNOT H37.00  ; #3腔体有清氦需求
AND H5.15  ; 腔体模式（0-正压 1-负压）
AND T2102  ; #3-1腔体破真空阈值到达延时（测试）
ANDNOT P_On
ORLD
OR D1135.10  ; #3腔体机构（清氦步）
LD D1135.11  ; #3腔体机构腔体顶升气缸下降（清氦步）
ANDNOT 803.02  ; #3腔体顶伸气缸上升位标志[0003.02]
AND 803.03  ; #3腔体顶伸气缸下降位标志[0003.03]
AND D1122.00  ; #3腔体机构平移气缸安全移动条件
ORLD
LD D1135.12  ; #3腔体机构腔体平移气缸到初始位（清氦步）
ANDNOT 802.14  ; #3腔体平移一级气缸缩回位标志[0002.14]
AND 802.15  ; #3腔体平移一级气缸伸出位标志[0002.15]
ANDNOT 803.00  ; #3腔体平移二级气缸缩回位标志[0003.00]
AND 803.01  ; #3腔体平移二级气缸伸出位标志[0003.01]
ORLD
OR D1135.13  ; #3腔体机构（清氦步）
OR D1135.14  ; #3腔体机构（清氦步）
LD D1135.15  ; #3腔体机构循环结束（清氦步）
AND P_On
ORLD
AND D1124.03  ; #3腔体机构自动循环运行中（清氦步）
OUT D1125.05  ; #3腔体机构步进条件（清氦步）

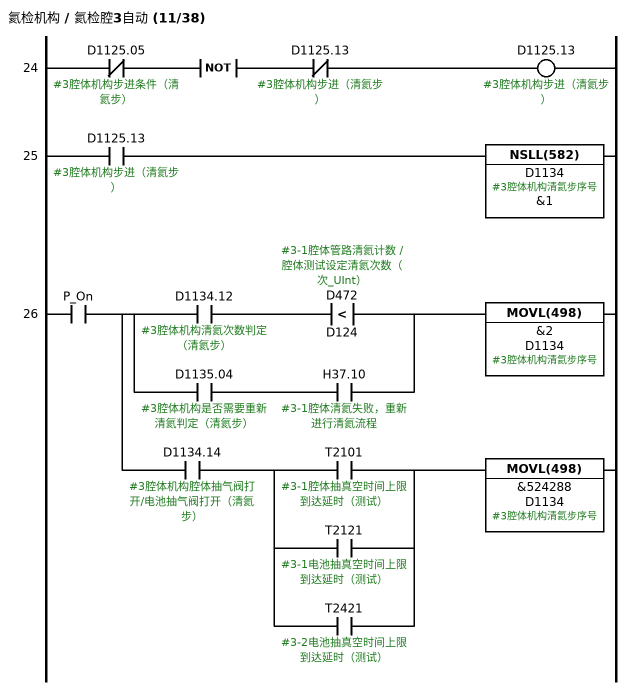
; rung 24
LDNOT D1125.05  ; #3腔体机构步进条件（清氦步）
NOT(520)
ANDNOT D1125.13  ; #3腔体机构步进（清氦步）
OUT D1125.13  ; #3腔体机构步进（清氦步）
; rung 25
LD D1125.13  ; #3腔体机构步进（清氦步）
NSLL(582) D1134 &1  ; #3腔体机构清氦步序号
; rung 26
LD P_On
OUT TR0
LD D1134.12  ; #3腔体机构清氦次数判定（清氦步）
AND<(310) D472 D124  ; #3-1腔体管路清氦计数, 腔体测试设定清氦次数（次_UInt）
LD D1135.04  ; #3腔体机构是否需要重新清氦判定（清氦步）
AND H37.10  ; #3-1腔体清氦失败，重新进行清氦流程  // 清氦失败，重新进行清氦
ORLD
ANDLD
MOVL(498) &2 D1134  ; #3腔体机构清氦步序号
LD TR0
AND D1134.14  ; #3腔体机构腔体抽气阀打开/电池抽气阀打开（清氦步）
LD T2101  ; #3-1腔体抽真空时间上限到达延时（测试）
OR T2121  ; #3-1电池抽真空时间上限到达延时（测试）
OR T2421  ; #3-2电池抽真空时间上限到达延时（测试）
ANDLD
MOVL(498) &524288 D1134  ; #3腔体机构清氦步序号  // 清氦过程腔体或电池抽气上限达到，均直接判定清氦完成，不进入氦检步序（跳转至D1075.03）

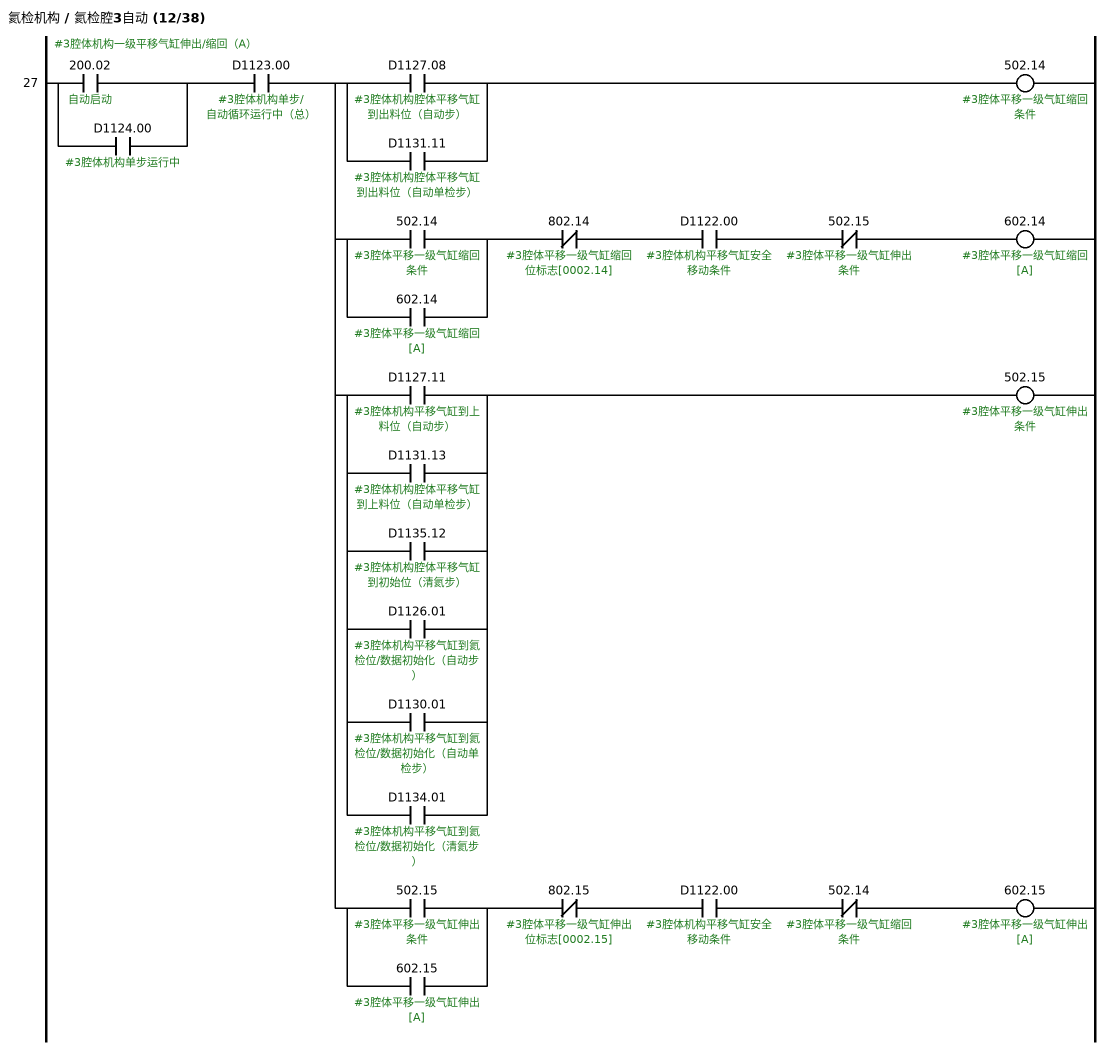
; rung 27: #3腔体机构一级平移气缸伸出/缩回（A）
LD 200.02  ; 自动启动
OR D1124.00  ; #3腔体机构单步运行中
AND D1123.00  ; #3腔体机构单步/自动循环运行中（总）
OUT TR0
LD D1127.08  ; #3腔体机构腔体平移气缸到出料位（自动步）
OR D1131.11  ; #3腔体机构腔体平移气缸到出料位（自动单检步）
ANDLD
OUT 502.14  ; #3腔体平移一级气缸缩回条件
LD TR0
LD 502.14  ; #3腔体平移一级气缸缩回条件
OR 602.14  ; #3腔体平移一级气缸缩回[A]
ANDLD
ANDNOT 802.14  ; #3腔体平移一级气缸缩回位标志[0002.14]
AND D1122.00  ; #3腔体机构平移气缸安全移动条件
ANDNOT 502.15  ; #3腔体平移一级气缸伸出条件
OUT 602.14  ; #3腔体平移一级气缸缩回[A]
LD TR0
LD D1127.11  ; #3腔体机构平移气缸到上料位（自动步）
OR D1131.13  ; #3腔体机构腔体平移气缸到上料位（自动单检步）
OR D1135.12  ; #3腔体机构腔体平移气缸到初始位（清氦步）
OR D1126.01  ; #3腔体机构平移气缸到氦检位/数据初始化（自动步）
OR D1130.01  ; #3腔体机构平移气缸到氦检位/数据初始化（自动单检步）
OR D1134.01  ; #3腔体机构平移气缸到氦检位/数据初始化（清氦步）
ANDLD
OUT 502.15  ; #3腔体平移一级气缸伸出条件
LD TR0
LD 502.15  ; #3腔体平移一级气缸伸出条件
OR 602.15  ; #3腔体平移一级气缸伸出[A]
ANDLD
ANDNOT 802.15  ; #3腔体平移一级气缸伸出位标志[0002.15]
AND D1122.00  ; #3腔体机构平移气缸安全移动条件
ANDNOT 502.14  ; #3腔体平移一级气缸缩回条件
OUT 602.15  ; #3腔体平移一级气缸伸出[A]

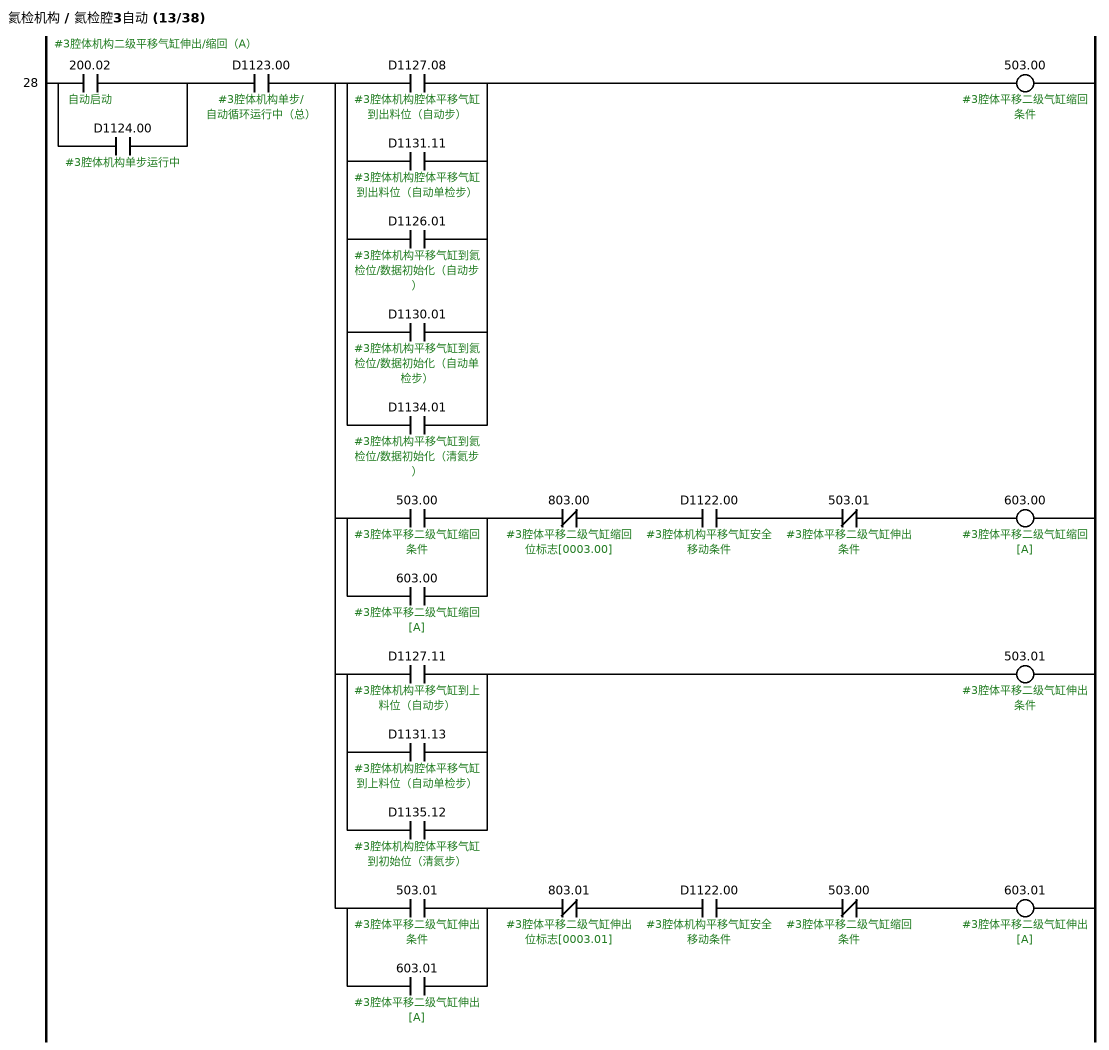
; rung 28: #3腔体机构二级平移气缸伸出/缩回（A）
LD 200.02  ; 自动启动
OR D1124.00  ; #3腔体机构单步运行中
AND D1123.00  ; #3腔体机构单步/自动循环运行中（总）
OUT TR0
LD D1127.08  ; #3腔体机构腔体平移气缸到出料位（自动步）
OR D1131.11  ; #3腔体机构腔体平移气缸到出料位（自动单检步）
OR D1126.01  ; #3腔体机构平移气缸到氦检位/数据初始化（自动步）
OR D1130.01  ; #3腔体机构平移气缸到氦检位/数据初始化（自动单检步）
OR D1134.01  ; #3腔体机构平移气缸到氦检位/数据初始化（清氦步）
ANDLD
OUT 503.00  ; #3腔体平移二级气缸缩回条件
LD TR0
LD 503.00  ; #3腔体平移二级气缸缩回条件
OR 603.00  ; #3腔体平移二级气缸缩回[A]
ANDLD
ANDNOT 803.00  ; #3腔体平移二级气缸缩回位标志[0003.00]
AND D1122.00  ; #3腔体机构平移气缸安全移动条件
ANDNOT 503.01  ; #3腔体平移二级气缸伸出条件
OUT 603.00  ; #3腔体平移二级气缸缩回[A]
LD TR0
LD D1127.11  ; #3腔体机构平移气缸到上料位（自动步）
OR D1131.13  ; #3腔体机构腔体平移气缸到上料位（自动单检步）
OR D1135.12  ; #3腔体机构腔体平移气缸到初始位（清氦步）
ANDLD
OUT 503.01  ; #3腔体平移二级气缸伸出条件
LD TR0
LD 503.01  ; #3腔体平移二级气缸伸出条件
OR 603.01  ; #3腔体平移二级气缸伸出[A]
ANDLD
ANDNOT 803.01  ; #3腔体平移二级气缸伸出位标志[0003.01]
AND D1122.00  ; #3腔体机构平移气缸安全移动条件
ANDNOT 503.00  ; #3腔体平移二级气缸缩回条件
OUT 603.01  ; #3腔体平移二级气缸伸出[A]

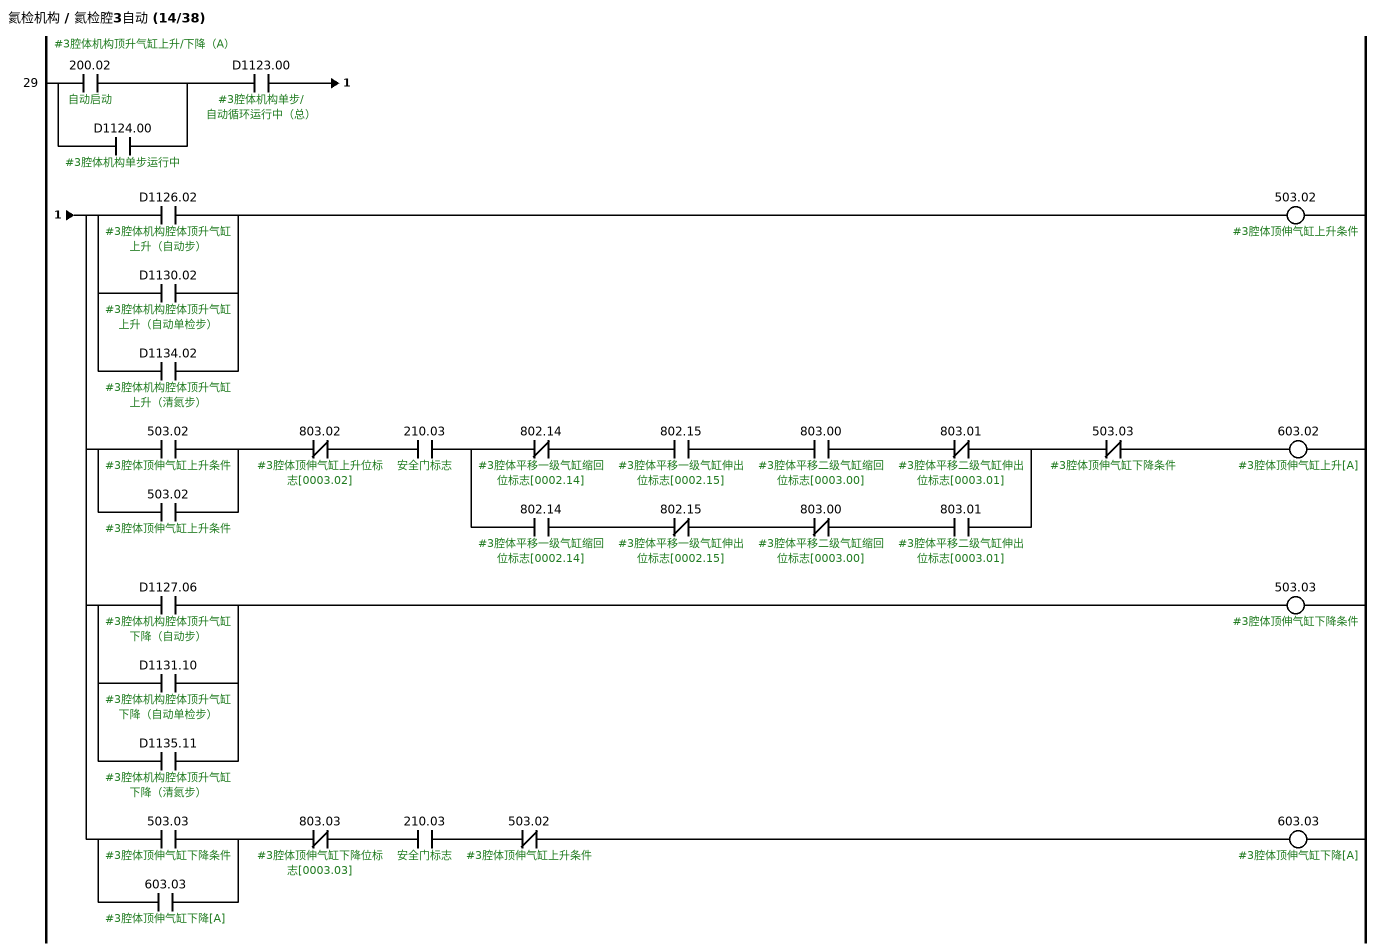
; rung 29: #3腔体机构顶升气缸上升/下降（A）
LD 200.02  ; 自动启动
OR D1124.00  ; #3腔体机构单步运行中
AND D1123.00  ; #3腔体机构单步/自动循环运行中（总）
OUT TR0
LD D1126.02  ; #3腔体机构腔体顶升气缸上升（自动步）
OR D1130.02  ; #3腔体机构腔体顶升气缸上升（自动单检步）
OR D1134.02  ; #3腔体机构腔体顶升气缸上升（清氦步）
ANDLD
OUT 503.02  ; #3腔体顶伸气缸上升条件
LD TR0
LD 503.02  ; #3腔体顶伸气缸上升条件
OR 503.02  ; #3腔体顶伸气缸上升条件
ANDLD
ANDNOT 803.02  ; #3腔体顶伸气缸上升位标志[0003.02]
AND 210.03  ; 安全门标志
LDNOT 802.14  ; #3腔体平移一级气缸缩回位标志[0002.14]
AND 802.15  ; #3腔体平移一级气缸伸出位标志[0002.15]
AND 803.00  ; #3腔体平移二级气缸缩回位标志[0003.00]
ANDNOT 803.01  ; #3腔体平移二级气缸伸出位标志[0003.01]
LD 802.14  ; #3腔体平移一级气缸缩回位标志[0002.14]
ANDNOT 802.15  ; #3腔体平移一级气缸伸出位标志[0002.15]
ANDNOT 803.00  ; #3腔体平移二级气缸缩回位标志[0003.00]
AND 803.01  ; #3腔体平移二级气缸伸出位标志[0003.01]
ORLD
ANDLD
ANDNOT 503.03  ; #3腔体顶伸气缸下降条件
OUT 603.02  ; #3腔体顶伸气缸上升[A]
LD TR0
LD D1127.06  ; #3腔体机构腔体顶升气缸下降（自动步）
OR D1131.10  ; #3腔体机构腔体顶升气缸下降（自动单检步）
OR D1135.11  ; #3腔体机构腔体顶升气缸下降（清氦步）
ANDLD
OUT 503.03  ; #3腔体顶伸气缸下降条件
LD TR0
LD 503.03  ; #3腔体顶伸气缸下降条件
OR 603.03  ; #3腔体顶伸气缸下降[A]
ANDLD
ANDNOT 803.03  ; #3腔体顶伸气缸下降位标志[0003.03]
AND 210.03  ; 安全门标志
ANDNOT 503.02  ; #3腔体顶伸气缸上升条件
OUT 603.03  ; #3腔体顶伸气缸下降[A]

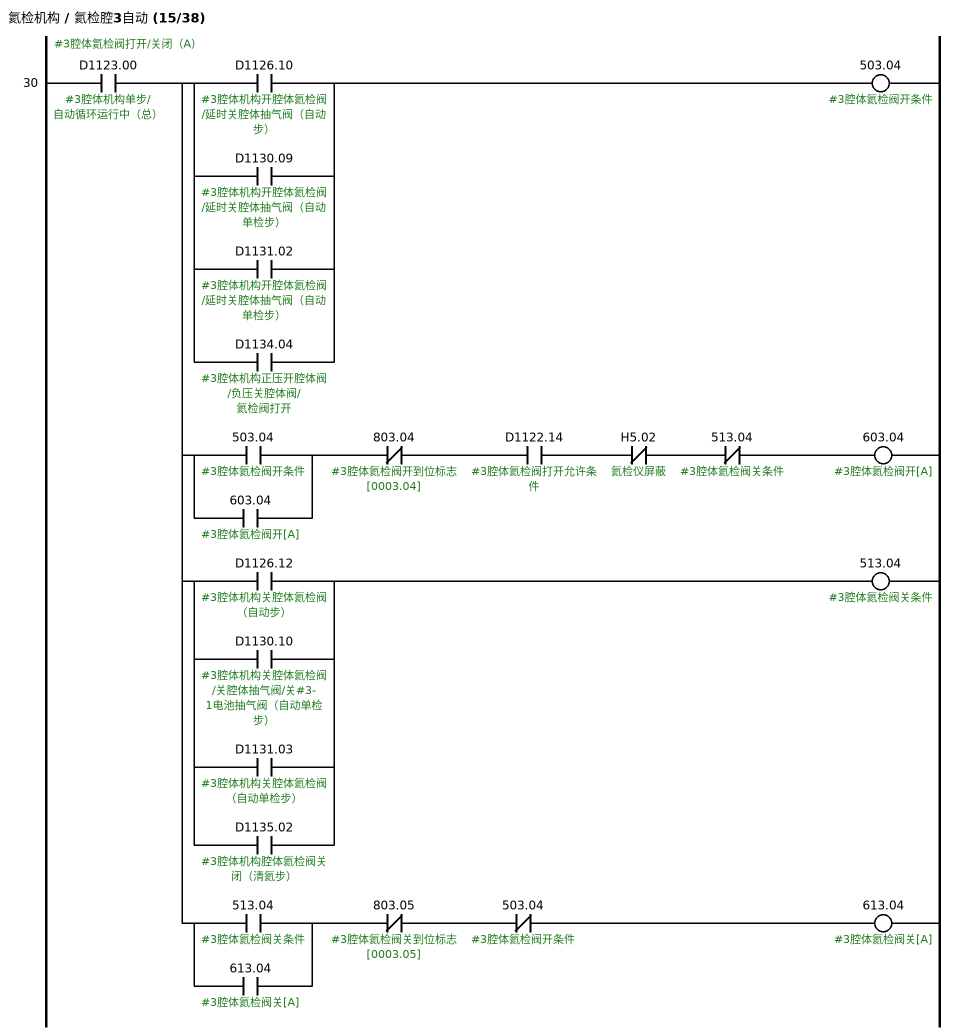
; rung 30: #3腔体氦检阀打开/关闭（A）
LD D1123.00  ; #3腔体机构单步/自动循环运行中（总）
OUT TR0
LD D1126.10  ; #3腔体机构开腔体氦检阀/延时关腔体抽气阀（自动步）
OR D1130.09  ; #3腔体机构开腔体氦检阀/延时关腔体抽气阀（自动单检步）
OR D1131.02  ; #3腔体机构开腔体氦检阀/延时关腔体抽气阀（自动单检步）
OR D1134.04  ; #3腔体机构正压开腔体阀/负压关腔体阀/氦检阀打开
ANDLD
OUT 503.04  ; #3腔体氦检阀开条件
LD TR0
LD 503.04  ; #3腔体氦检阀开条件
OR 603.04  ; #3腔体氦检阀开[A]
ANDLD
ANDNOT 803.04  ; #3腔体氦检阀开到位标志[0003.04]
AND D1122.14  ; #3腔体氦检阀打开允许条件
ANDNOT H5.02  ; 氦检仪屏蔽
ANDNOT 513.04  ; #3腔体氦检阀关条件
OUT 603.04  ; #3腔体氦检阀开[A]
LD TR0
LD D1126.12  ; #3腔体机构关腔体氦检阀（自动步）
OR D1130.10  ; #3腔体机构关腔体氦检阀/关腔体抽气阀/关#3-1电池抽气阀（自动单检步）
OR D1131.03  ; #3腔体机构关腔体氦检阀（自动单检步）
OR D1135.02  ; #3腔体机构腔体氦检阀关闭（清氦步）
ANDLD
OUT 513.04  ; #3腔体氦检阀关条件
LD TR0
LD 513.04  ; #3腔体氦检阀关条件
OR 613.04  ; #3腔体氦检阀关[A]
ANDLD
ANDNOT 803.05  ; #3腔体氦检阀关到位标志[0003.05]
ANDNOT 503.04  ; #3腔体氦检阀开条件
OUT 613.04  ; #3腔体氦检阀关[A]

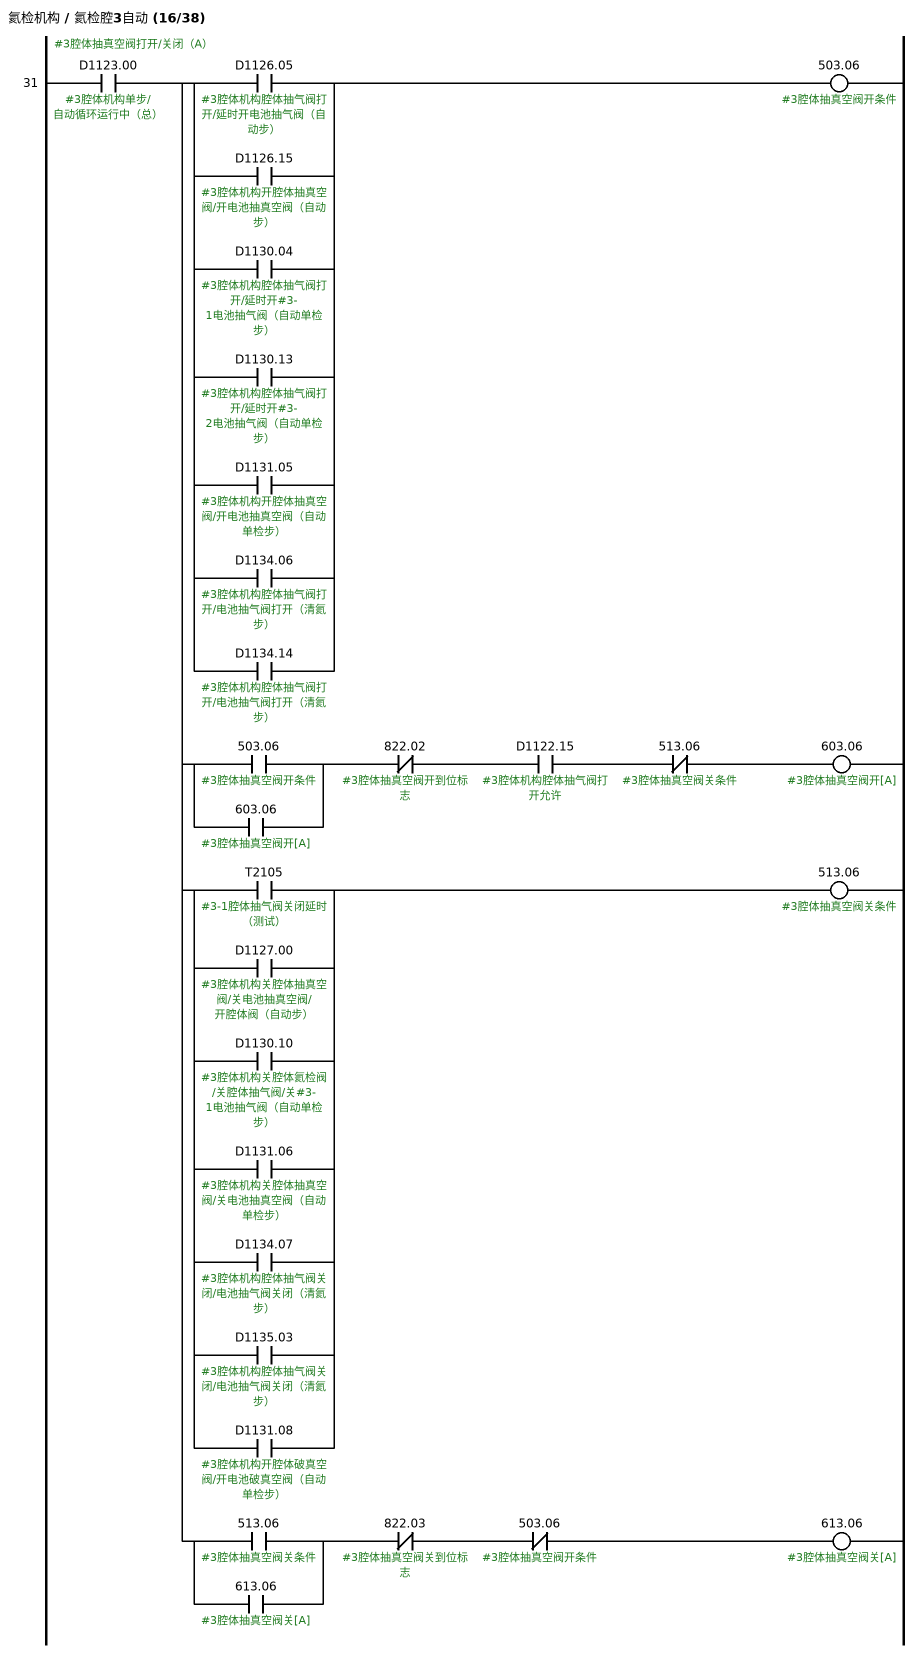
; rung 31: #3腔体抽真空阀打开/关闭（A）
LD D1123.00  ; #3腔体机构单步/自动循环运行中（总）
OUT TR0
LD D1126.05  ; #3腔体机构腔体抽气阀打开/延时开电池抽气阀（自动步）
OR D1126.15  ; #3腔体机构开腔体抽真空阀/开电池抽真空阀（自动步）
OR D1130.04  ; #3腔体机构腔体抽气阀打开/延时开#3-1电池抽气阀（自动单检步）
OR D1130.13  ; #3腔体机构腔体抽气阀打开/延时开#3-2电池抽气阀（自动单检步）
OR D1131.05  ; #3腔体机构开腔体抽真空阀/开电池抽真空阀（自动单检步）
OR D1134.06  ; #3腔体机构腔体抽气阀打开/电池抽气阀打开（清氦步）
OR D1134.14  ; #3腔体机构腔体抽气阀打开/电池抽气阀打开（清氦步）
ANDLD
OUT 503.06  ; #3腔体抽真空阀开条件
LD TR0
LD 503.06  ; #3腔体抽真空阀开条件
OR 603.06  ; #3腔体抽真空阀开[A]
ANDLD
ANDNOT 822.02  ; #3腔体抽真空阀开到位标志
AND D1122.15  ; #3腔体机构腔体抽气阀打开允许
ANDNOT 513.06  ; #3腔体抽真空阀关条件
OUT 603.06  ; #3腔体抽真空阀开[A]
LD TR0
LD T2105  ; #3-1腔体抽气阀关闭延时（测试）
OR D1127.00  ; #3腔体机构关腔体抽真空阀/关电池抽真空阀/开腔体阀（自动步）
OR D1130.10  ; #3腔体机构关腔体氦检阀/关腔体抽气阀/关#3-1电池抽气阀（自动单检步）
OR D1131.06  ; #3腔体机构关腔体抽真空阀/关电池抽真空阀（自动单检步）
OR D1134.07  ; #3腔体机构腔体抽气阀关闭/电池抽气阀关闭（清氦步）
OR D1135.03  ; #3腔体机构腔体抽气阀关闭/电池抽气阀关闭（清氦步）
OR D1131.08  ; #3腔体机构开腔体破真空阀/开电池破真空阀（自动单检步）
ANDLD
OUT 513.06  ; #3腔体抽真空阀关条件
LD TR0
LD 513.06  ; #3腔体抽真空阀关条件
OR 613.06  ; #3腔体抽真空阀关[A]
ANDLD
ANDNOT 822.03  ; #3腔体抽真空阀关到位标志
ANDNOT 503.06  ; #3腔体抽真空阀开条件
OUT 613.06  ; #3腔体抽真空阀关[A]

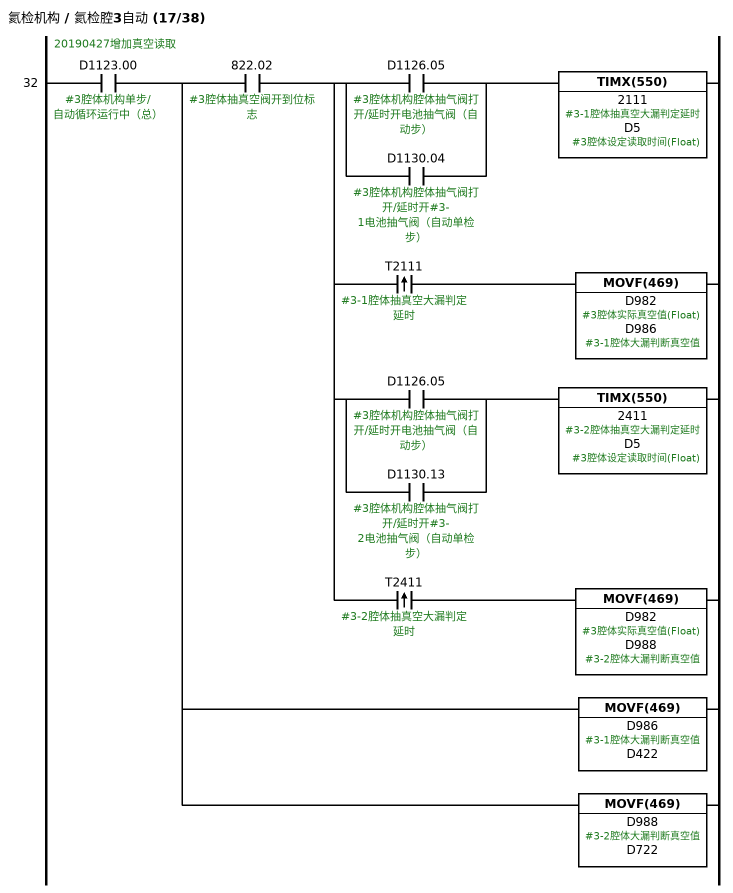
; rung 32: 20190427增加真空读取
LD D1123.00  ; #3腔体机构单步/自动循环运行中（总）
OUT TR0
AND 822.02  ; #3腔体抽真空阀开到位标志
OUT TR1
LD D1126.05  ; #3腔体机构腔体抽气阀打开/延时开电池抽气阀（自动步）
OR D1130.04  ; #3腔体机构腔体抽气阀打开/延时开#3-1电池抽气阀（自动单检步）
ANDLD
TIMX(550) 2111 D5  ; #3腔体设定读取时间(Float), #3-1腔体抽真空大漏判定延时
LD TR1
@AND T2111  ; #3-1腔体抽真空大漏判定延时
MOVF(469) D982 D986  ; #3腔体实际真空值(Float), #3-1腔体大漏判断真空值
LD TR1
LD D1126.05  ; #3腔体机构腔体抽气阀打开/延时开电池抽气阀（自动步）
OR D1130.13  ; #3腔体机构腔体抽气阀打开/延时开#3-2电池抽气阀（自动单检步）
ANDLD
TIMX(550) 2411 D5  ; #3腔体设定读取时间(Float), #3-2腔体抽真空大漏判定延时
LD TR1
@AND T2411  ; #3-2腔体抽真空大漏判定延时
MOVF(469) D982 D988  ; #3腔体实际真空值(Float), #3-2腔体大漏判断真空值
LD TR0
MOVF(469) D986 D422  ; #3-1腔体大漏判断真空值
MOVF(469) D988 D722  ; #3-2腔体大漏判断真空值

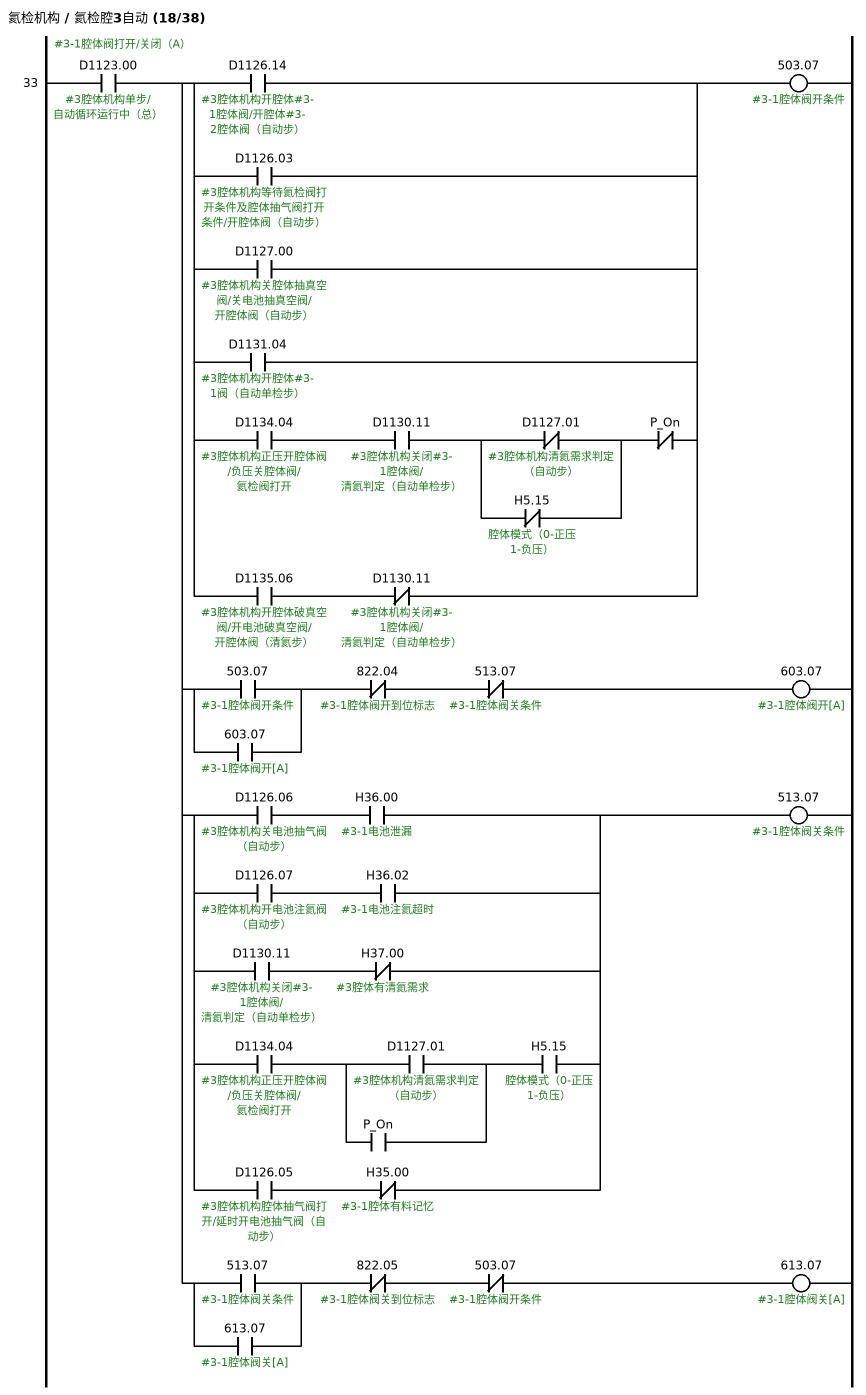
; rung 33: #3-1腔体阀打开/关闭（A）
LD D1123.00  ; #3腔体机构单步/自动循环运行中（总）
OUT TR0
LD D1126.14  ; #3腔体机构开腔体#3-1腔体阀/开腔体#3-2腔体阀（自动步）
OR D1126.03  ; #3腔体机构等待氦检阀打开条件及腔体抽气阀打开条件/开腔体阀（自动步）
OR D1127.00  ; #3腔体机构关腔体抽真空阀/关电池抽真空阀/开腔体阀（自动步）
OR D1131.04  ; #3腔体机构开腔体#3-1阀（自动单检步）
LD D1134.04  ; #3腔体机构正压开腔体阀/负压关腔体阀/氦检阀打开
AND D1130.11  ; #3腔体机构关闭#3-1腔体阀/清氦判定（自动单检步）
LDNOT D1127.01  ; #3腔体机构清氦需求判定（自动步）
ORNOT H5.15  ; 腔体模式（0-正压 1-负压）
ANDLD
ANDNOT P_On
ORLD
LD D1135.06  ; #3腔体机构开腔体破真空阀/开电池破真空阀/开腔体阀（清氦步）
ANDNOT D1130.11  ; #3腔体机构关闭#3-1腔体阀/清氦判定（自动单检步）
ORLD
ANDLD
OUT 503.07  ; #3-1腔体阀开条件
LD TR0
LD 503.07  ; #3-1腔体阀开条件
OR 603.07  ; #3-1腔体阀开[A]
ANDLD
ANDNOT 822.04  ; #3-1腔体阀开到位标志
ANDNOT 513.07  ; #3-1腔体阀关条件
OUT 603.07  ; #3-1腔体阀开[A]
LD TR0
LD D1126.06  ; #3腔体机构关电池抽气阀（自动步）
AND H36.00  ; #3-1电池泄漏
LD D1126.07  ; #3腔体机构开电池注氦阀（自动步）
AND H36.02  ; #3-1电池注氦超时
ORLD
LD D1130.11  ; #3腔体机构关闭#3-1腔体阀/清氦判定（自动单检步）
ANDNOT H37.00  ; #3腔体有清氦需求
ORLD
LD D1134.04  ; #3腔体机构正压开腔体阀/负压关腔体阀/氦检阀打开
LD D1127.01  ; #3腔体机构清氦需求判定（自动步）
OR P_On
ANDLD
AND H5.15  ; 腔体模式（0-正压 1-负压）
ORLD
LD D1126.05  ; #3腔体机构腔体抽气阀打开/延时开电池抽气阀（自动步）  // #1-1无料时不测试
ANDNOT H35.00  ; #3-1腔体有料记忆
ORLD
ANDLD
OUT 513.07  ; #3-1腔体阀关条件
LD TR0
LD 513.07  ; #3-1腔体阀关条件
OR 613.07  ; #3-1腔体阀关[A]
ANDLD
ANDNOT 822.05  ; #3-1腔体阀关到位标志
ANDNOT 503.07  ; #3-1腔体阀开条件
OUT 613.07  ; #3-1腔体阀关[A]

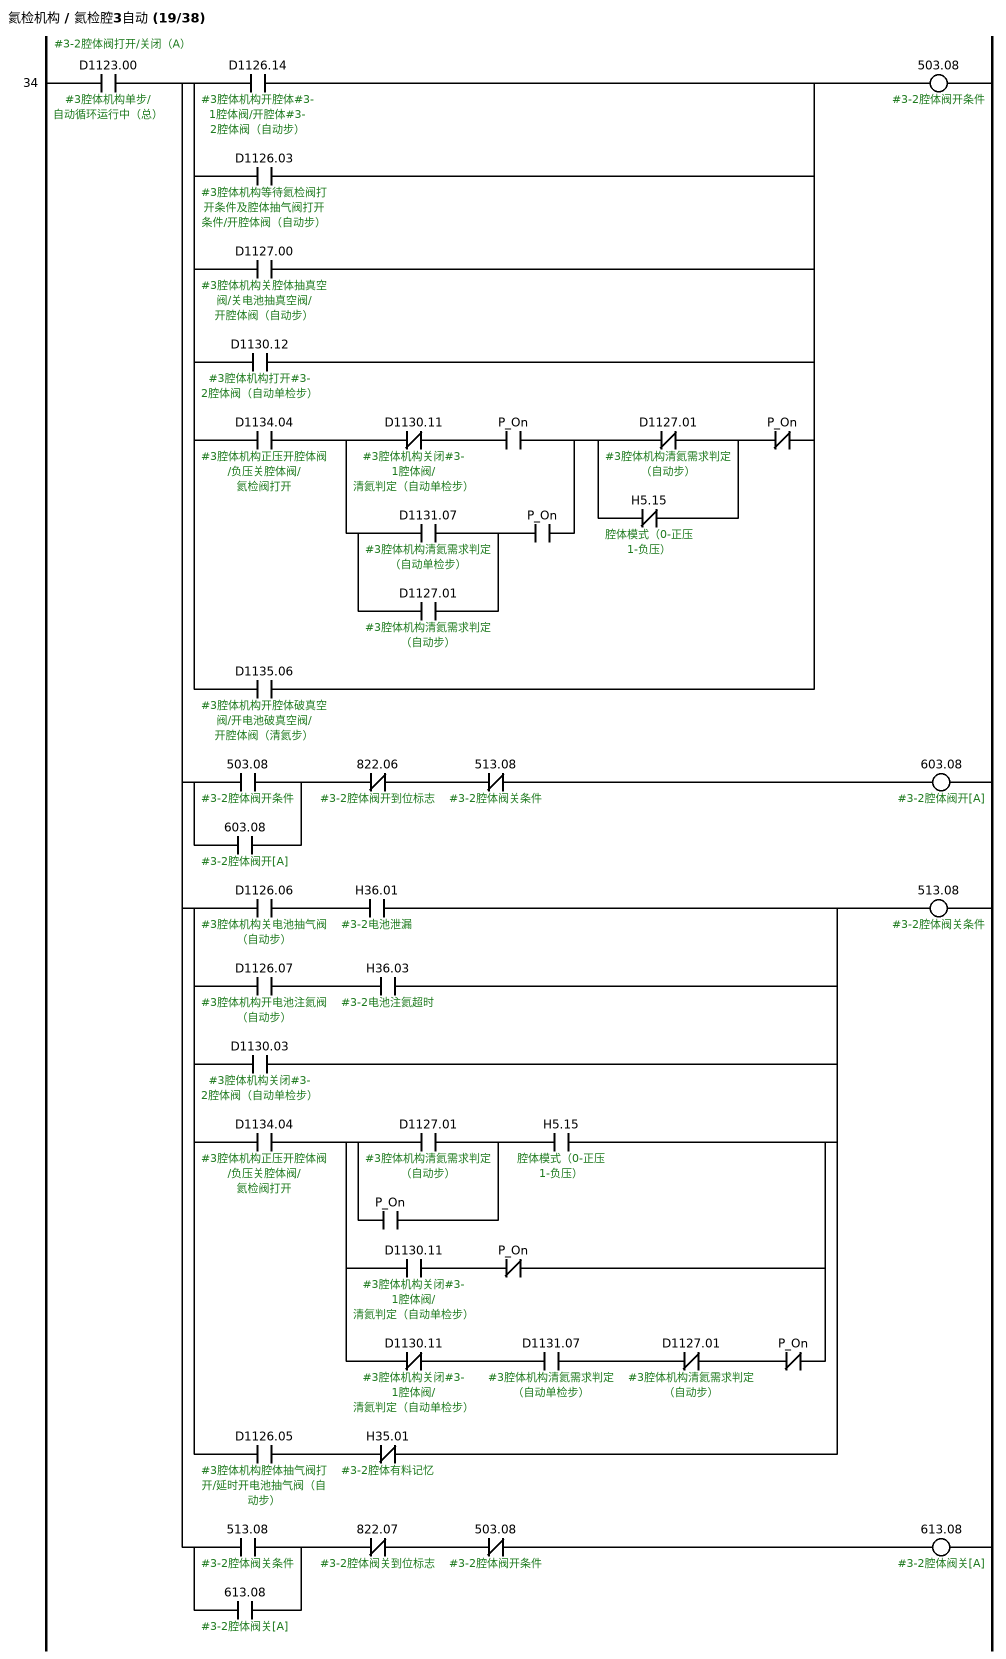
; rung 34: #3-2腔体阀打开/关闭（A）
LD D1123.00  ; #3腔体机构单步/自动循环运行中（总）
OUT TR0
LD D1126.14  ; #3腔体机构开腔体#3-1腔体阀/开腔体#3-2腔体阀（自动步）
OR D1126.03  ; #3腔体机构等待氦检阀打开条件及腔体抽气阀打开条件/开腔体阀（自动步）
OR D1127.00  ; #3腔体机构关腔体抽真空阀/关电池抽真空阀/开腔体阀（自动步）
OR D1130.12  ; #3腔体机构打开#3-2腔体阀（自动单检步）
LD D1134.04  ; #3腔体机构正压开腔体阀/负压关腔体阀/氦检阀打开
LDNOT D1130.11  ; #3腔体机构关闭#3-1腔体阀/清氦判定（自动单检步）
AND P_On
LD D1131.07  ; #3腔体机构清氦需求判定（自动单检步）
OR D1127.01  ; #3腔体机构清氦需求判定（自动步）
AND P_On
ORLD
ANDLD
LDNOT D1127.01  ; #3腔体机构清氦需求判定（自动步）
ORNOT H5.15  ; 腔体模式（0-正压 1-负压）
ANDLD
ANDNOT P_On
ORLD
OR D1135.06  ; #3腔体机构开腔体破真空阀/开电池破真空阀/开腔体阀（清氦步）
ANDLD
OUT 503.08  ; #3-2腔体阀开条件
LD TR0
LD 503.08  ; #3-2腔体阀开条件
OR 603.08  ; #3-2腔体阀开[A]
ANDLD
ANDNOT 822.06  ; #3-2腔体阀开到位标志
ANDNOT 513.08  ; #3-2腔体阀关条件
OUT 603.08  ; #3-2腔体阀开[A]
LD TR0
LD D1126.06  ; #3腔体机构关电池抽气阀（自动步）
AND H36.01  ; #3-2电池泄漏
LD D1126.07  ; #3腔体机构开电池注氦阀（自动步）
AND H36.03  ; #3-2电池注氦超时
ORLD
OR D1130.03  ; #3腔体机构关闭#3-2腔体阀（自动单检步）
LD D1134.04  ; #3腔体机构正压开腔体阀/负压关腔体阀/氦检阀打开
LD D1127.01  ; #3腔体机构清氦需求判定（自动步）
OR P_On
AND H5.15  ; 腔体模式（0-正压 1-负压）
LD D1130.11  ; #3腔体机构关闭#3-1腔体阀/清氦判定（自动单检步）
ANDNOT P_On
ORLD
LDNOT D1130.11  ; #3腔体机构关闭#3-1腔体阀/清氦判定（自动单检步）
AND D1131.07  ; #3腔体机构清氦需求判定（自动单检步）
ANDNOT D1127.01  ; #3腔体机构清氦需求判定（自动步）
ANDNOT P_On
ORLD
ANDLD
ORLD
LD D1126.05  ; #3腔体机构腔体抽气阀打开/延时开电池抽气阀（自动步）  // #1-2无料时不测试
ANDNOT H35.01  ; #3-2腔体有料记忆
ORLD
ANDLD
OUT 513.08  ; #3-2腔体阀关条件
LD TR0
LD 513.08  ; #3-2腔体阀关条件
OR 613.08  ; #3-2腔体阀关[A]
ANDLD
ANDNOT 822.07  ; #3-2腔体阀关到位标志
ANDNOT 503.08  ; #3-2腔体阀开条件
OUT 613.08  ; #3-2腔体阀关[A]

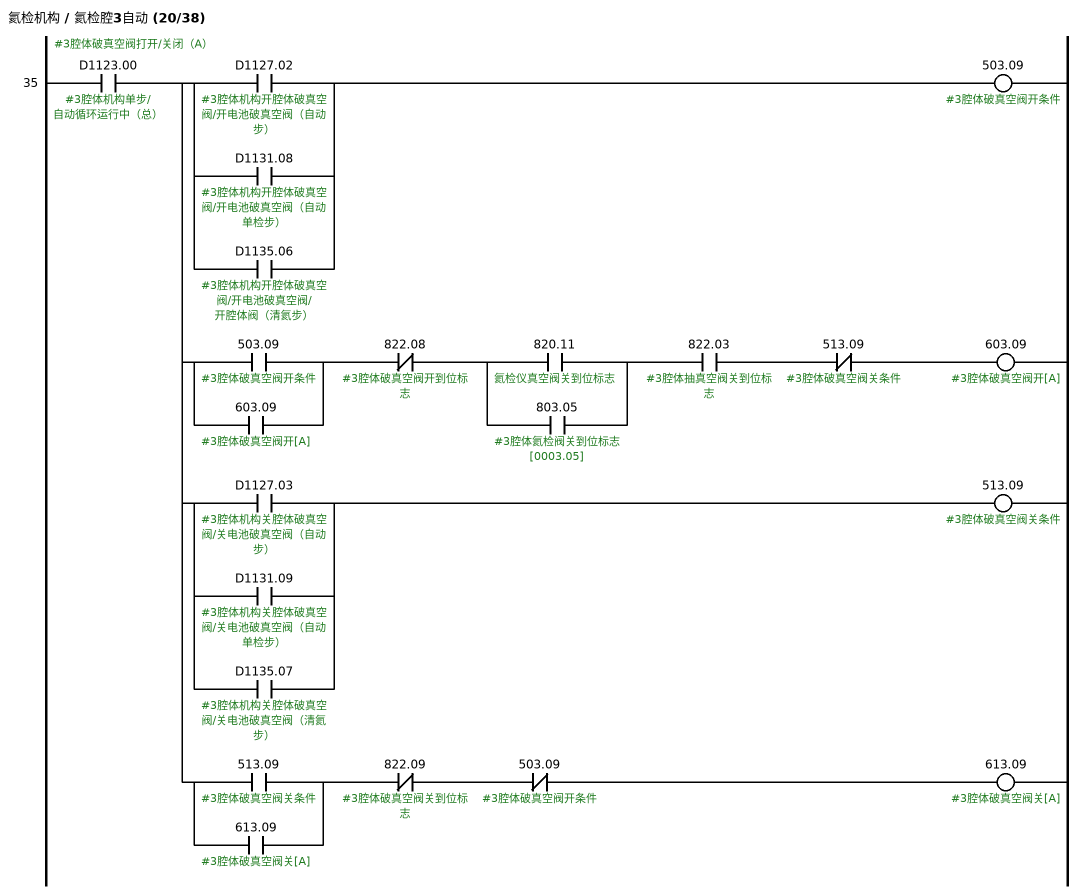
; rung 35: #3腔体破真空阀打开/关闭（A）
LD D1123.00  ; #3腔体机构单步/自动循环运行中（总）
OUT TR0
LD D1127.02  ; #3腔体机构开腔体破真空阀/开电池破真空阀（自动步）
OR D1131.08  ; #3腔体机构开腔体破真空阀/开电池破真空阀（自动单检步）
OR D1135.06  ; #3腔体机构开腔体破真空阀/开电池破真空阀/开腔体阀（清氦步）
ANDLD
OUT 503.09  ; #3腔体破真空阀开条件
LD TR0
LD 503.09  ; #3腔体破真空阀开条件
OR 603.09  ; #3腔体破真空阀开[A]
ANDLD
ANDNOT 822.08  ; #3腔体破真空阀开到位标志
LD 820.11  ; 氦检仪真空阀关到位标志
OR 803.05  ; #3腔体氦检阀关到位标志[0003.05]
ANDLD
AND 822.03  ; #3腔体抽真空阀关到位标志
ANDNOT 513.09  ; #3腔体破真空阀关条件
OUT 603.09  ; #3腔体破真空阀开[A]
LD TR0
LD D1127.03  ; #3腔体机构关腔体破真空阀/关电池破真空阀（自动步）
OR D1131.09  ; #3腔体机构关腔体破真空阀/关电池破真空阀（自动单检步）
OR D1135.07  ; #3腔体机构关腔体破真空阀/关电池破真空阀（清氦步）
ANDLD
OUT 513.09  ; #3腔体破真空阀关条件
LD TR0
LD 513.09  ; #3腔体破真空阀关条件
OR 613.09  ; #3腔体破真空阀关[A]
ANDLD
ANDNOT 822.09  ; #3腔体破真空阀关到位标志
ANDNOT 503.09  ; #3腔体破真空阀开条件
OUT 613.09  ; #3腔体破真空阀关[A]

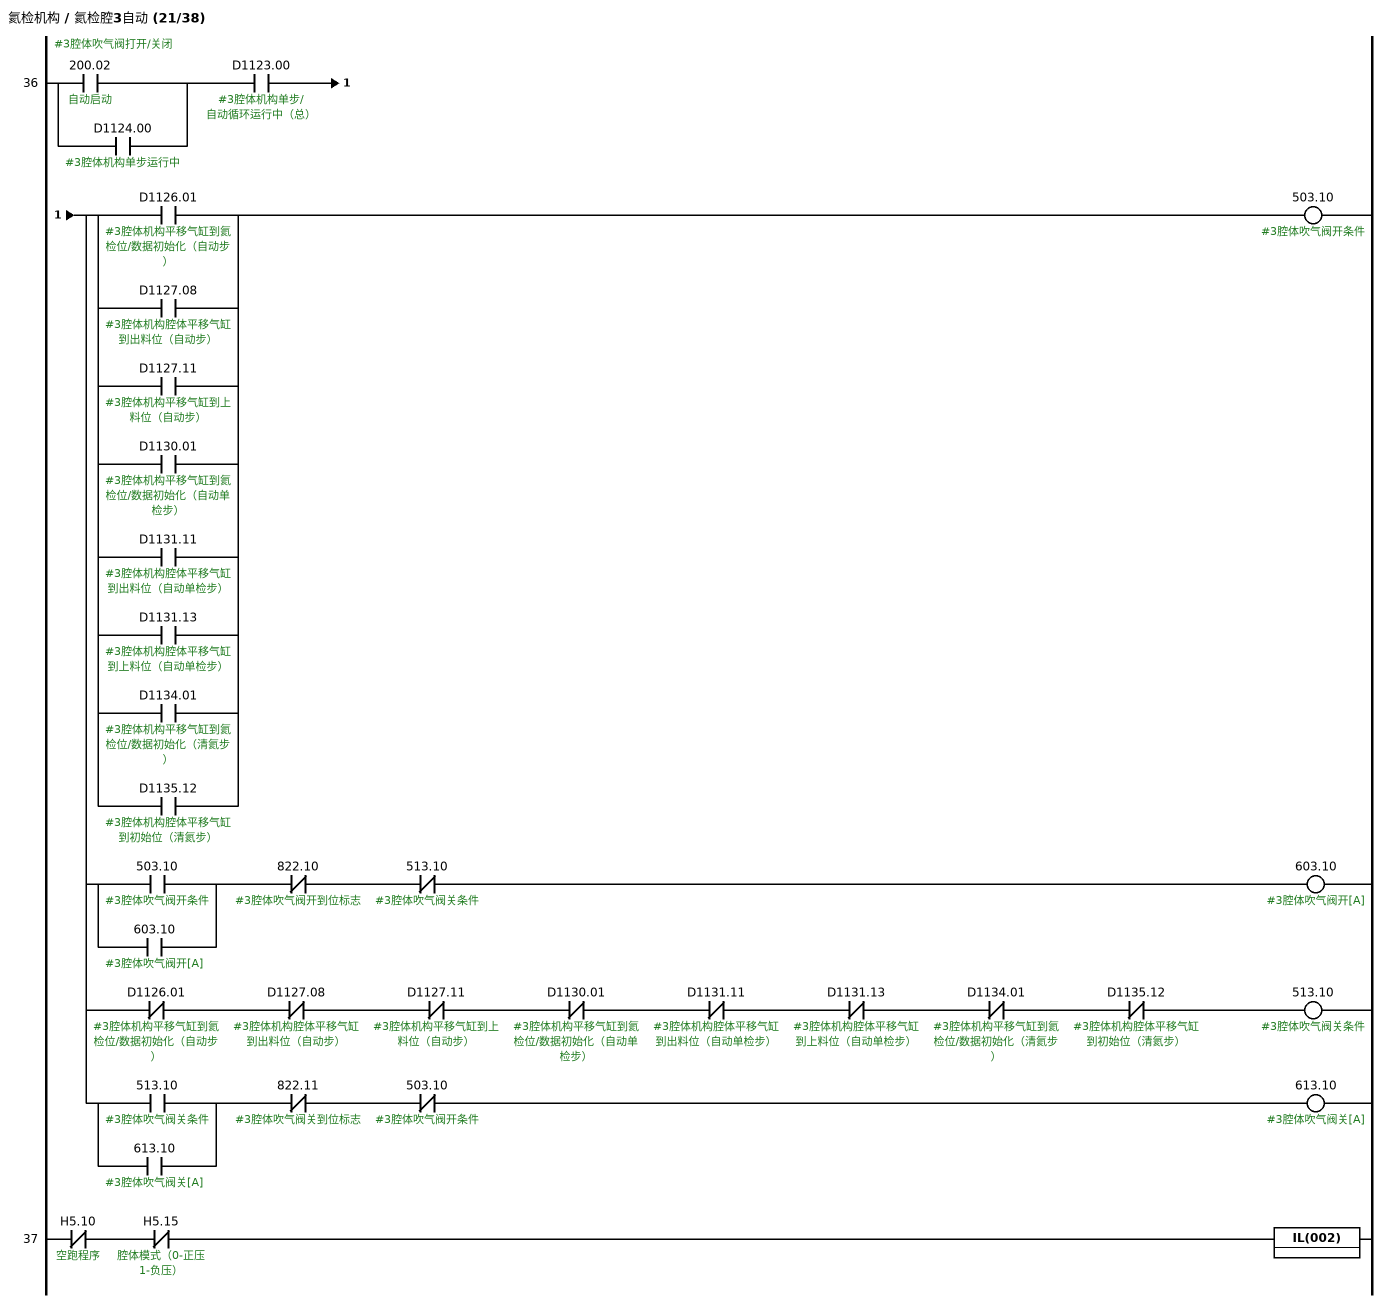
; rung 36: #3腔体吹气阀打开/关闭
LD 200.02  ; 自动启动
OR D1124.00  ; #3腔体机构单步运行中
AND D1123.00  ; #3腔体机构单步/自动循环运行中（总）
OUT TR0
LD D1126.01  ; #3腔体机构平移气缸到氦检位/数据初始化（自动步）
OR D1127.08  ; #3腔体机构腔体平移气缸到出料位（自动步）
OR D1127.11  ; #3腔体机构平移气缸到上料位（自动步）
OR D1130.01  ; #3腔体机构平移气缸到氦检位/数据初始化（自动单检步）
OR D1131.11  ; #3腔体机构腔体平移气缸到出料位（自动单检步）
OR D1131.13  ; #3腔体机构腔体平移气缸到上料位（自动单检步）
OR D1134.01  ; #3腔体机构平移气缸到氦检位/数据初始化（清氦步）
OR D1135.12  ; #3腔体机构腔体平移气缸到初始位（清氦步）
ANDLD
OUT 503.10  ; #3腔体吹气阀开条件
LD TR0
LD 503.10  ; #3腔体吹气阀开条件
OR 603.10  ; #3腔体吹气阀开[A]
ANDLD
ANDNOT 822.10  ; #3腔体吹气阀开到位标志
ANDNOT 513.10  ; #3腔体吹气阀关条件
OUT 603.10  ; #3腔体吹气阀开[A]
LD TR0
ANDNOT D1126.01  ; #3腔体机构平移气缸到氦检位/数据初始化（自动步）
ANDNOT D1127.08  ; #3腔体机构腔体平移气缸到出料位（自动步）
ANDNOT D1127.11  ; #3腔体机构平移气缸到上料位（自动步）
ANDNOT D1130.01  ; #3腔体机构平移气缸到氦检位/数据初始化（自动单检步）
ANDNOT D1131.11  ; #3腔体机构腔体平移气缸到出料位（自动单检步）
ANDNOT D1131.13  ; #3腔体机构腔体平移气缸到上料位（自动单检步）
ANDNOT D1134.01  ; #3腔体机构平移气缸到氦检位/数据初始化（清氦步）
ANDNOT D1135.12  ; #3腔体机构腔体平移气缸到初始位（清氦步）
OUT 513.10  ; #3腔体吹气阀关条件
LD TR0
LD 513.10  ; #3腔体吹气阀关条件
OR 613.10  ; #3腔体吹气阀关[A]
ANDLD
ANDNOT 822.11  ; #3腔体吹气阀关到位标志
ANDNOT 503.10  ; #3腔体吹气阀开条件
OUT 613.10  ; #3腔体吹气阀关[A]
; rung 37
LDNOT H5.10  ; 空跑程序
ANDNOT H5.15  ; 腔体模式（0-正压 1-负压）
IL(002)

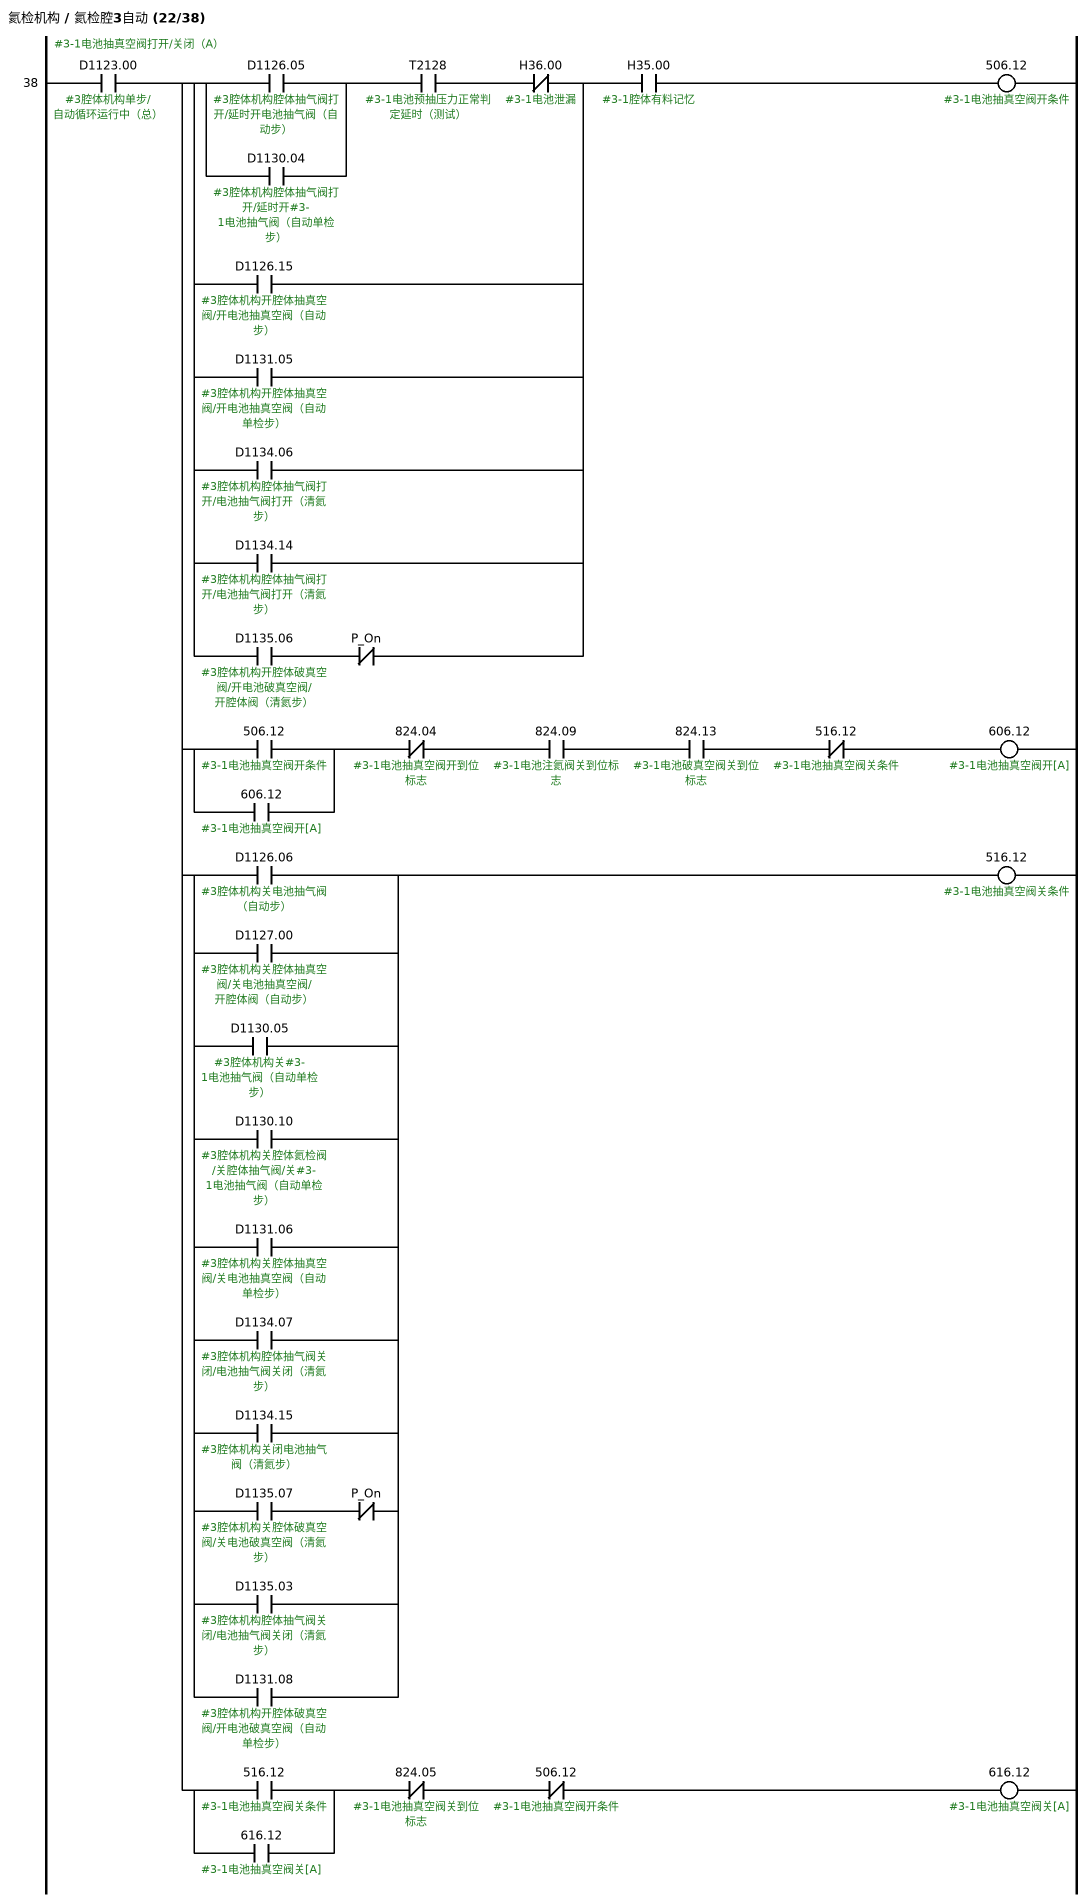
; rung 38: #3-1电池抽真空阀打开/关闭（A）
LD D1123.00  ; #3腔体机构单步/自动循环运行中（总）
OUT TR0
LD D1126.05  ; #3腔体机构腔体抽气阀打开/延时开电池抽气阀（自动步）
OR D1130.04  ; #3腔体机构腔体抽气阀打开/延时开#3-1电池抽气阀（自动单检步）
AND T2128  ; #3-1电池预抽压力正常判定延时（测试）
ANDNOT H36.00  ; #3-1电池泄漏
OR D1126.15  ; #3腔体机构开腔体抽真空阀/开电池抽真空阀（自动步）
OR D1131.05  ; #3腔体机构开腔体抽真空阀/开电池抽真空阀（自动单检步）
OR D1134.06  ; #3腔体机构腔体抽气阀打开/电池抽气阀打开（清氦步）
OR D1134.14  ; #3腔体机构腔体抽气阀打开/电池抽气阀打开（清氦步）
LD D1135.06  ; #3腔体机构开腔体破真空阀/开电池破真空阀/开腔体阀（清氦步）
ANDNOT P_On
ORLD
ANDLD
AND H35.00  ; #3-1腔体有料记忆
OUT 506.12  ; #3-1电池抽真空阀开条件
LD TR0
LD 506.12  ; #3-1电池抽真空阀开条件
OR 606.12  ; #3-1电池抽真空阀开[A]
ANDLD
ANDNOT 824.04  ; #3-1电池抽真空阀开到位标志
AND 824.09  ; #3-1电池注氦阀关到位标志
AND 824.13  ; #3-1电池破真空阀关到位标志
ANDNOT 516.12  ; #3-1电池抽真空阀关条件
OUT 606.12  ; #3-1电池抽真空阀开[A]
LD TR0
LD D1126.06  ; #3腔体机构关电池抽气阀（自动步）
OR D1127.00  ; #3腔体机构关腔体抽真空阀/关电池抽真空阀/开腔体阀（自动步）
OR D1130.05  ; #3腔体机构关#3-1电池抽气阀（自动单检步）
OR D1130.10  ; #3腔体机构关腔体氦检阀/关腔体抽气阀/关#3-1电池抽气阀（自动单检步）
OR D1131.06  ; #3腔体机构关腔体抽真空阀/关电池抽真空阀（自动单检步）
OR D1134.07  ; #3腔体机构腔体抽气阀关闭/电池抽气阀关闭（清氦步）
OR D1134.15  ; #3腔体机构关闭电池抽气阀（清氦步）
LD D1135.07  ; #3腔体机构关腔体破真空阀/关电池破真空阀（清氦步）
ANDNOT P_On
ORLD
OR D1135.03  ; #3腔体机构腔体抽气阀关闭/电池抽气阀关闭（清氦步）
OR D1131.08  ; #3腔体机构开腔体破真空阀/开电池破真空阀（自动单检步）
ANDLD
OUT 516.12  ; #3-1电池抽真空阀关条件
LD TR0
LD 516.12  ; #3-1电池抽真空阀关条件
OR 616.12  ; #3-1电池抽真空阀关[A]
ANDLD
ANDNOT 824.05  ; #3-1电池抽真空阀关到位标志
ANDNOT 506.12  ; #3-1电池抽真空阀开条件
OUT 616.12  ; #3-1电池抽真空阀关[A]

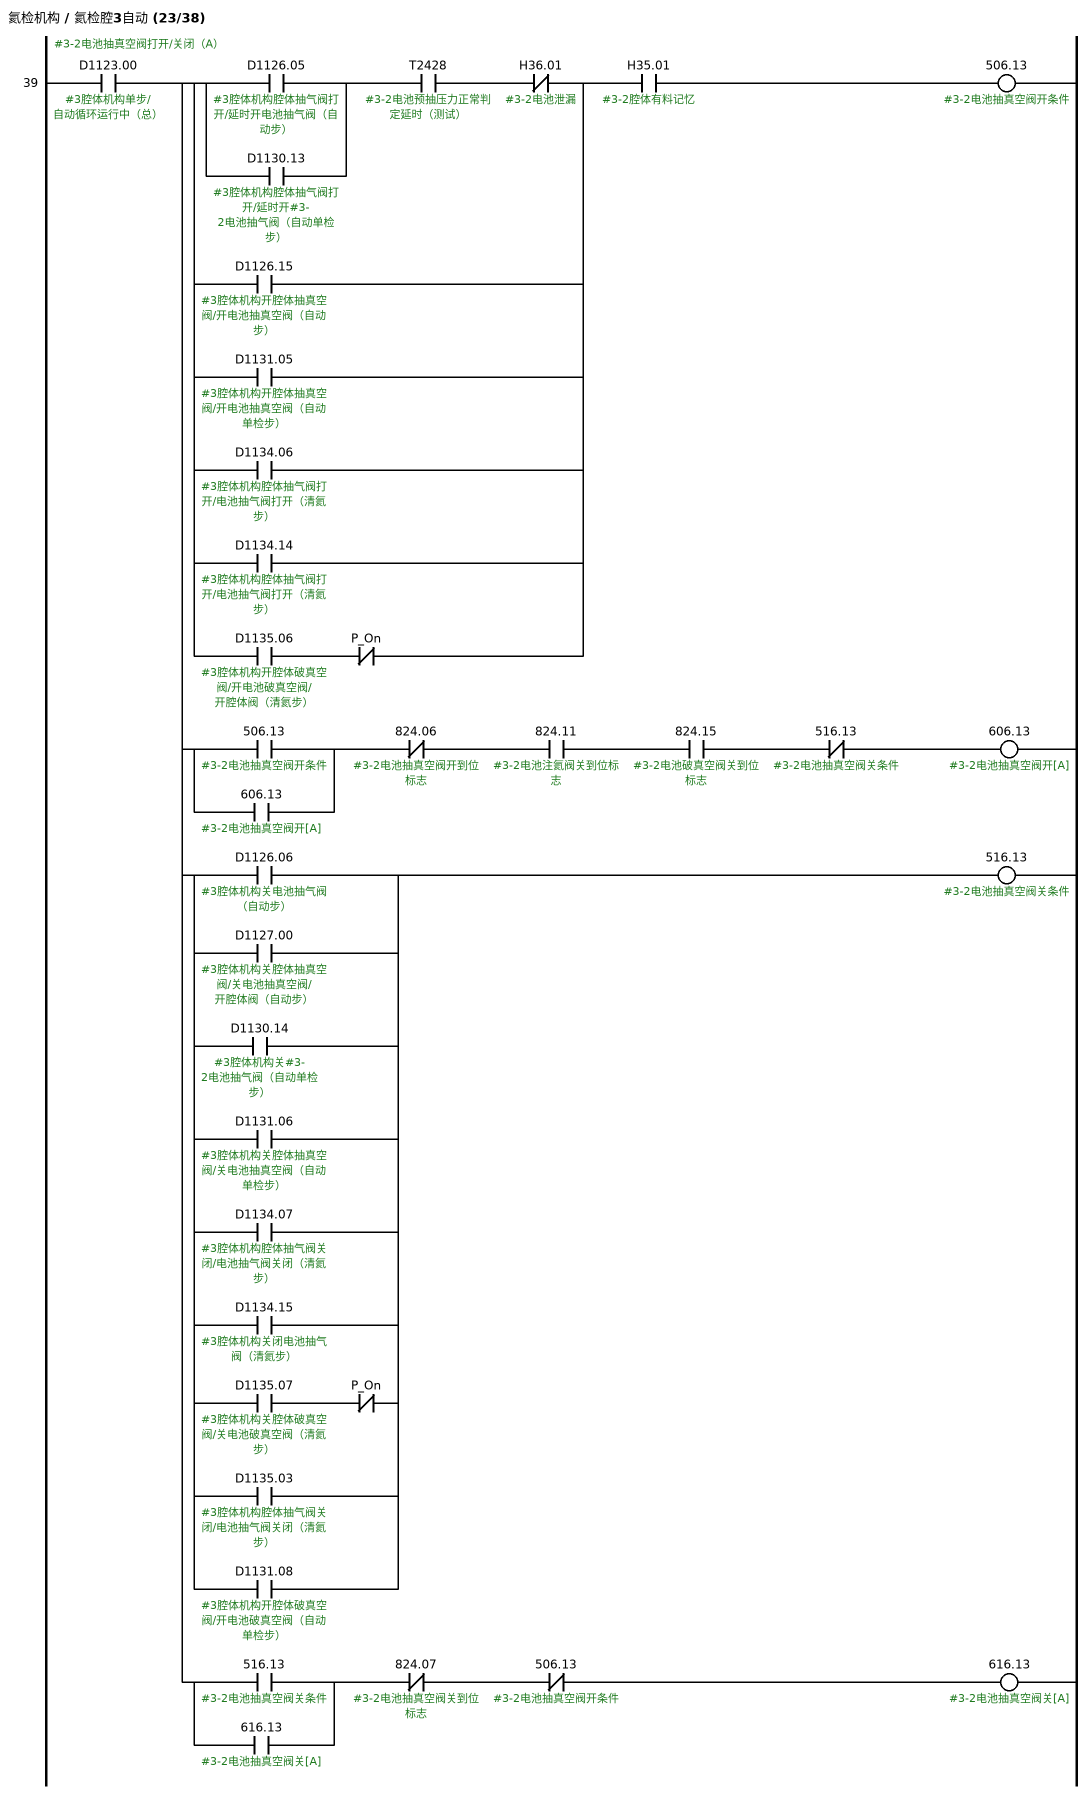
; rung 39: #3-2电池抽真空阀打开/关闭（A）
LD D1123.00  ; #3腔体机构单步/自动循环运行中（总）
OUT TR0
LD D1126.05  ; #3腔体机构腔体抽气阀打开/延时开电池抽气阀（自动步）
OR D1130.13  ; #3腔体机构腔体抽气阀打开/延时开#3-2电池抽气阀（自动单检步）
AND T2428  ; #3-2电池预抽压力正常判定延时（测试）
ANDNOT H36.01  ; #3-2电池泄漏
OR D1126.15  ; #3腔体机构开腔体抽真空阀/开电池抽真空阀（自动步）
OR D1131.05  ; #3腔体机构开腔体抽真空阀/开电池抽真空阀（自动单检步）
OR D1134.06  ; #3腔体机构腔体抽气阀打开/电池抽气阀打开（清氦步）
OR D1134.14  ; #3腔体机构腔体抽气阀打开/电池抽气阀打开（清氦步）
LD D1135.06  ; #3腔体机构开腔体破真空阀/开电池破真空阀/开腔体阀（清氦步）
ANDNOT P_On
ORLD
ANDLD
AND H35.01  ; #3-2腔体有料记忆
OUT 506.13  ; #3-2电池抽真空阀开条件
LD TR0
LD 506.13  ; #3-2电池抽真空阀开条件
OR 606.13  ; #3-2电池抽真空阀开[A]
ANDLD
ANDNOT 824.06  ; #3-2电池抽真空阀开到位标志
AND 824.11  ; #3-2电池注氦阀关到位标志
AND 824.15  ; #3-2电池破真空阀关到位标志
ANDNOT 516.13  ; #3-2电池抽真空阀关条件
OUT 606.13  ; #3-2电池抽真空阀开[A]
LD TR0
LD D1126.06  ; #3腔体机构关电池抽气阀（自动步）
OR D1127.00  ; #3腔体机构关腔体抽真空阀/关电池抽真空阀/开腔体阀（自动步）
OR D1130.14  ; #3腔体机构关#3-2电池抽气阀（自动单检步）
OR D1131.06  ; #3腔体机构关腔体抽真空阀/关电池抽真空阀（自动单检步）
OR D1134.07  ; #3腔体机构腔体抽气阀关闭/电池抽气阀关闭（清氦步）
OR D1134.15  ; #3腔体机构关闭电池抽气阀（清氦步）
LD D1135.07  ; #3腔体机构关腔体破真空阀/关电池破真空阀（清氦步）
ANDNOT P_On
ORLD
OR D1135.03  ; #3腔体机构腔体抽气阀关闭/电池抽气阀关闭（清氦步）
OR D1131.08  ; #3腔体机构开腔体破真空阀/开电池破真空阀（自动单检步）
ANDLD
OUT 516.13  ; #3-2电池抽真空阀关条件
LD TR0
LD 516.13  ; #3-2电池抽真空阀关条件
OR 616.13  ; #3-2电池抽真空阀关[A]
ANDLD
ANDNOT 824.07  ; #3-2电池抽真空阀关到位标志
ANDNOT 506.13  ; #3-2电池抽真空阀开条件
OUT 616.13  ; #3-2电池抽真空阀关[A]

